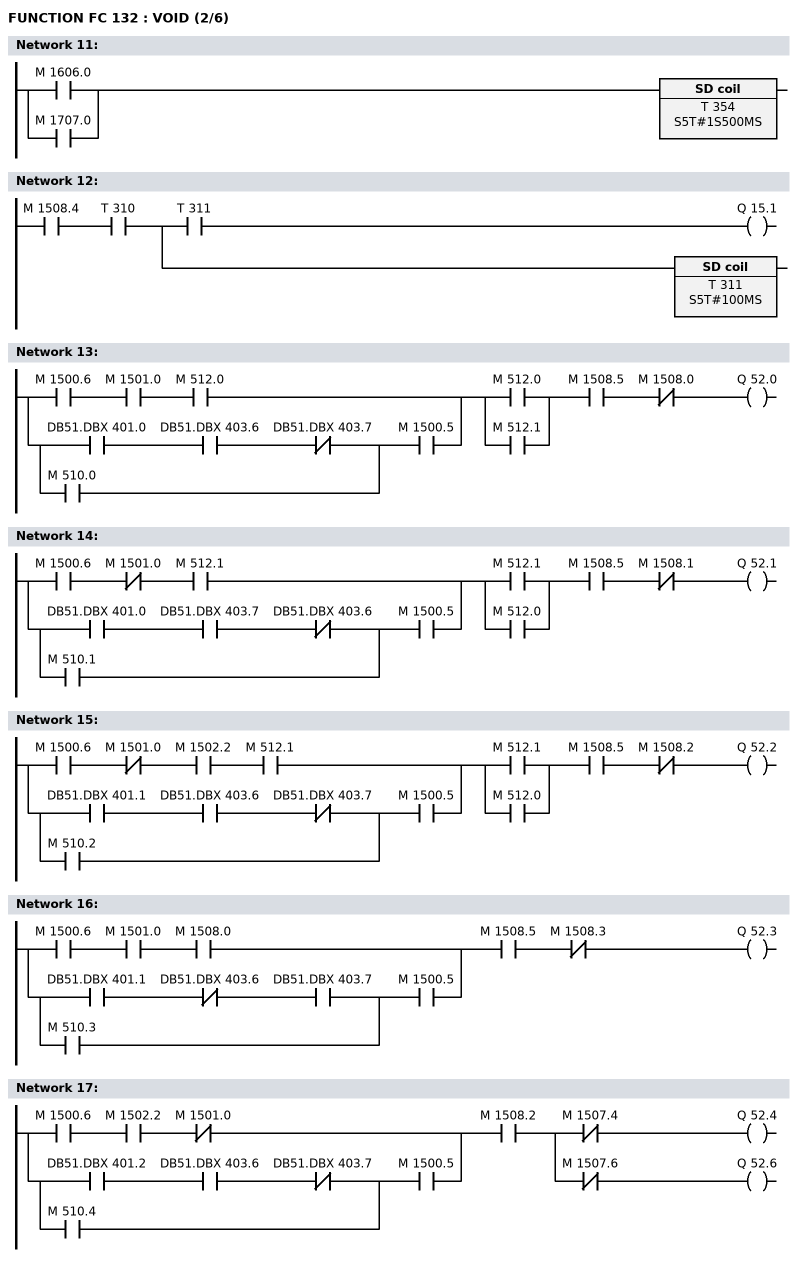

      O     M   1606.0;
      O     M   1707.0;
      L     S5T#1S500MS;
      SD    T    354;
NETWORK
TITLE =

      A     M   1508.4;
      A     T    310;
      =     L      0.0;
      A     L      0.0;
      A     T    311;
      =     Q     15.1;
      A     L      0.0;
      BLD   102;
      L     S5T#100MS;
      SD    T    311;
NETWORK
TITLE =

      A(    ;
      A     M   1500.6;
      A     M   1501.0;
      A     M    512.0;
      O     ;
      A(    ;
      A     DB51.DBX  401.0;
      A     DB51.DBX  403.6;
      AN    DB51.DBX  403.7;
      O     M    510.0;
      )     ;
      A     M   1500.5;
      )     ;
      A(    ;
      O     M    512.0;
      O     M    512.1;
      )     ;
      A     M   1508.5;
      AN    M   1508.0;
      =     Q     52.0;
NETWORK
TITLE =

      A(    ;
      A     M   1500.6;
      AN    M   1501.0;
      A     M    512.1;
      O     ;
      A(    ;
      A     DB51.DBX  401.0;
      A     DB51.DBX  403.7;
      AN    DB51.DBX  403.6;
      O     M    510.1;
      )     ;
      A     M   1500.5;
      )     ;
      A(    ;
      O     M    512.1;
      O     M    512.0;
      )     ;
      A     M   1508.5;
      AN    M   1508.1;
      =     Q     52.1;
NETWORK
TITLE =

      A(    ;
      A     M   1500.6;
      AN    M   1501.0;
      A     M   1502.2;
      A     M    512.1;
      O     ;
      A(    ;
      A     DB51.DBX  401.1;
      A     DB51.DBX  403.6;
      AN    DB51.DBX  403.7;
      O     M    510.2;
      )     ;
      A     M   1500.5;
      )     ;
      A(    ;
      O     M    512.1;
      O     M    512.0;
      )     ;
      A     M   1508.5;
      AN    M   1508.2;
      =     Q     52.2;
NETWORK
TITLE =

      A(    ;
      A     M   1500.6;
      A     M   1501.0;
      A     M   1508.0;
      O     ;
      A(    ;
      A     DB51.DBX  401.1;
      AN    DB51.DBX  403.6;
      A     DB51.DBX  403.7;
      O     M    510.3;
      )     ;
      A     M   1500.5;
      )     ;
      A     M   1508.5;
      AN    M   1508.3;
      =     Q     52.3;
NETWORK
TITLE =

      A(    ;
      A     M   1500.6;
      A     M   1502.2;
      AN    M   1501.0;
      O     ;
      A(    ;
      A     DB51.DBX  401.2;
      A     DB51.DBX  403.6;
      AN    DB51.DBX  403.7;
      O     M    510.4;
      )     ;
      A     M   1500.5;
      )     ;
      A     M   1508.2;
      =     L      0.0;
      A     L      0.0;
      AN    M   1507.4;
      =     Q     52.4;
      A     L      0.0;
      AN    M   1507.6;
      =     Q     52.6;
NETWORK
TITLE =
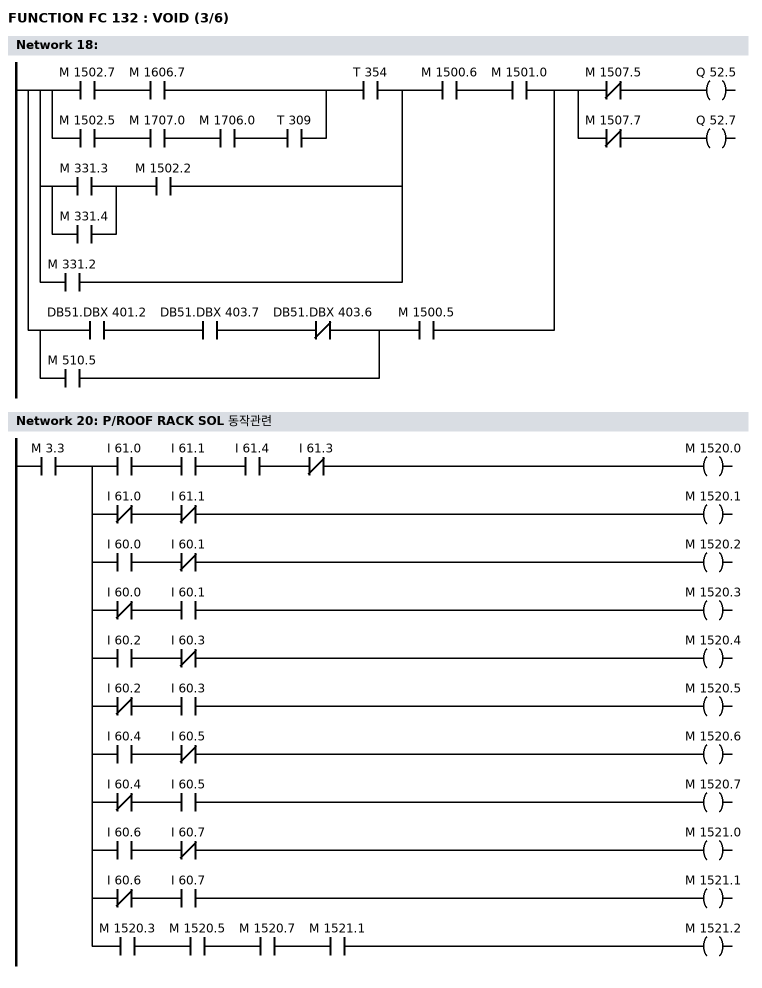

      A(    ;
      A(    ;
      A     M   1502.7;
      A     M   1606.7;
      O     ;
      A     M   1502.5;
      A     M   1707.0;
      A     M   1706.0;
      A     T    309;
      )     ;
      A     T    354;
      O     ;
      A(    ;
      O     M    331.3;
      O     M    331.4;
      )     ;
      A     M   1502.2;
      O     M    331.2;
      )     ;
      A     M   1500.6;
      A     M   1501.0;
      O     ;
      A(    ;
      A     DB51.DBX  401.2;
      A     DB51.DBX  403.7;
      AN    DB51.DBX  403.6;
      O     M    510.5;
      )     ;
      A     M   1500.5;
      =     L      0.0;
      A     L      0.0;
      AN    M   1507.5;
      =     Q     52.5;
      A     L      0.0;
      AN    M   1507.7;
      =     Q     52.7;
NETWORK
TITLE =

NETWORK
TITLE =P/ROOF RACK SOL 동작관련

      A     M      3.3;
      =     L      0.0;
      A     L      0.0;
      A     I     61.0;
      A     I     61.1;
      A     I     61.4;
      AN    I     61.3;
      =     M   1520.0;
      A     L      0.0;
      AN    I     61.0;
      AN    I     61.1;
      =     M   1520.1;
      A     L      0.0;
      A     I     60.0;
      AN    I     60.1;
      =     M   1520.2;
      A     L      0.0;
      AN    I     60.0;
      A     I     60.1;
      =     M   1520.3;
      A     L      0.0;
      A     I     60.2;
      AN    I     60.3;
      =     M   1520.4;
      A     L      0.0;
      AN    I     60.2;
      A     I     60.3;
      =     M   1520.5;
      A     L      0.0;
      A     I     60.4;
      AN    I     60.5;
      =     M   1520.6;
      A     L      0.0;
      AN    I     60.4;
      A     I     60.5;
      =     M   1520.7;
      A     L      0.0;
      A     I     60.6;
      AN    I     60.7;
      =     M   1521.0;
      A     L      0.0;
      AN    I     60.6;
      A     I     60.7;
      =     M   1521.1;
      A     L      0.0;
      A     M   1520.3;
      A     M   1520.5;
      A     M   1520.7;
      A     M   1521.1;
      =     M   1521.2;
NETWORK
TITLE =
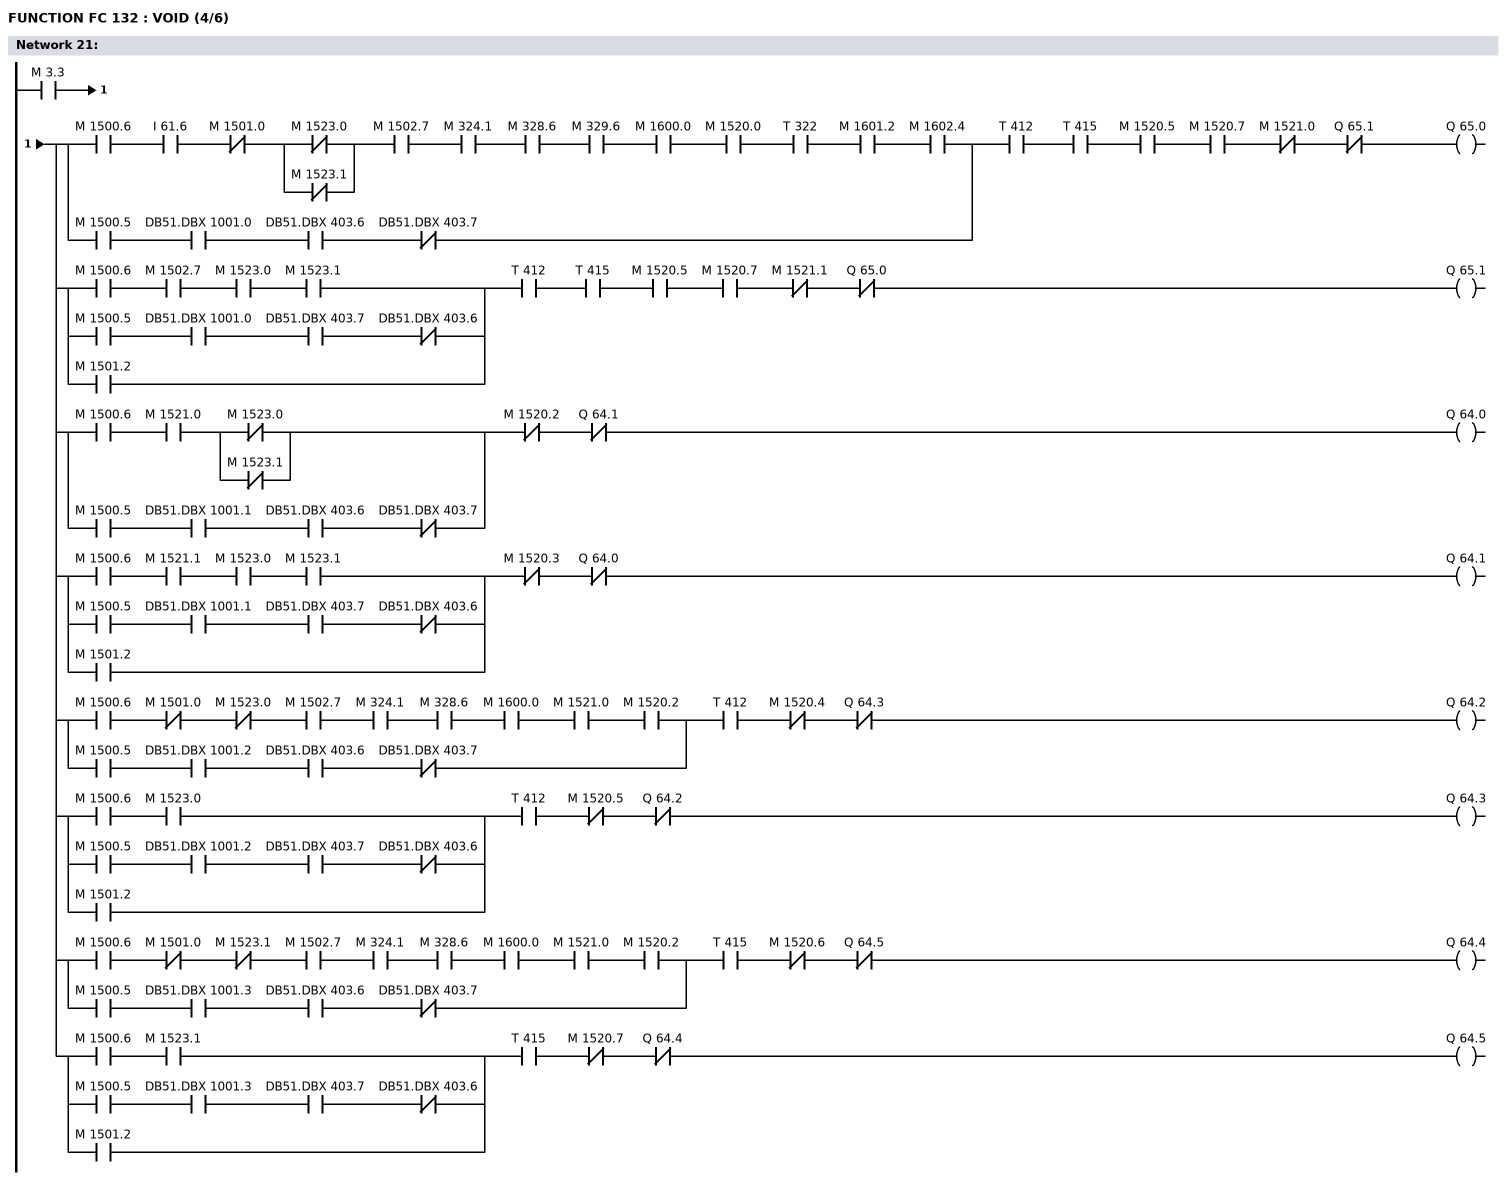

      A     M      3.3;
      =     L      0.0;
      A     L      0.0;
      A(    ;
      A     M   1500.6;
      A     I     61.6;
      AN    M   1501.0;
      A(    ;
      ON    M   1523.0;
      ON    M   1523.1;
      )     ;
      A     M   1502.7;
      A     M    324.1;
      A     M    328.6;
      A     M    329.6;
      A     M   1600.0;
      A     M   1520.0;
      A     T    322;
      A     M   1601.2;
      A     M   1602.4;
      O     ;
      A     M   1500.5;
      A     DB51.DBX 1001.0;
      A     DB51.DBX  403.6;
      AN    DB51.DBX  403.7;
      )     ;
      A     T    412;
      A     T    415;
      A     M   1520.5;
      A     M   1520.7;
      AN    M   1521.0;
      AN    Q     65.1;
      =     Q     65.0;
      A     L      0.0;
      A(    ;
      A     M   1500.6;
      A     M   1502.7;
      A     M   1523.0;
      A     M   1523.1;
      O     ;
      A     M   1500.5;
      A     DB51.DBX 1001.0;
      A     DB51.DBX  403.7;
      AN    DB51.DBX  403.6;
      O     M   1501.2;
      )     ;
      A     T    412;
      A     T    415;
      A     M   1520.5;
      A     M   1520.7;
      AN    M   1521.1;
      AN    Q     65.0;
      =     Q     65.1;
      A     L      0.0;
      A(    ;
      A     M   1500.6;
      A     M   1521.0;
      A(    ;
      ON    M   1523.0;
      ON    M   1523.1;
      )     ;
      O     ;
      A     M   1500.5;
      A     DB51.DBX 1001.1;
      A     DB51.DBX  403.6;
      AN    DB51.DBX  403.7;
      )     ;
      AN    M   1520.2;
      AN    Q     64.1;
      =     Q     64.0;
      A     L      0.0;
      A(    ;
      A     M   1500.6;
      A     M   1521.1;
      A     M   1523.0;
      A     M   1523.1;
      O     ;
      A     M   1500.5;
      A     DB51.DBX 1001.1;
      A     DB51.DBX  403.7;
      AN    DB51.DBX  403.6;
      O     M   1501.2;
      )     ;
      AN    M   1520.3;
      AN    Q     64.0;
      =     Q     64.1;
      A     L      0.0;
      A(    ;
      A     M   1500.6;
      AN    M   1501.0;
      AN    M   1523.0;
      A     M   1502.7;
      A     M    324.1;
      A     M    328.6;
      A     M   1600.0;
      A     M   1521.0;
      A     M   1520.2;
      O     ;
      A     M   1500.5;
      A     DB51.DBX 1001.2;
      A     DB51.DBX  403.6;
      AN    DB51.DBX  403.7;
      )     ;
      A     T    412;
      AN    M   1520.4;
      AN    Q     64.3;
      =     Q     64.2;
      A     L      0.0;
      A(    ;
      A     M   1500.6;
      A     M   1523.0;
      O     ;
      A     M   1500.5;
      A     DB51.DBX 1001.2;
      A     DB51.DBX  403.7;
      AN    DB51.DBX  403.6;
      O     M   1501.2;
      )     ;
      A     T    412;
      AN    M   1520.5;
      AN    Q     64.2;
      =     Q     64.3;
      A     L      0.0;
      A(    ;
      A     M   1500.6;
      AN    M   1501.0;
      AN    M   1523.1;
      A     M   1502.7;
      A     M    324.1;
      A     M    328.6;
      A     M   1600.0;
      A     M   1521.0;
      A     M   1520.2;
      O     ;
      A     M   1500.5;
      A     DB51.DBX 1001.3;
      A     DB51.DBX  403.6;
      AN    DB51.DBX  403.7;
      )     ;
      A     T    415;
      AN    M   1520.6;
      AN    Q     64.5;
      =     Q     64.4;
      A     L      0.0;
      A(    ;
      A     M   1500.6;
      A     M   1523.1;
      O     ;
      A     M   1500.5;
      A     DB51.DBX 1001.3;
      A     DB51.DBX  403.7;
      AN    DB51.DBX  403.6;
      O     M   1501.2;
      )     ;
      A     T    415;
      AN    M   1520.7;
      AN    Q     64.4;
      =     Q     64.5;
NETWORK
TITLE =
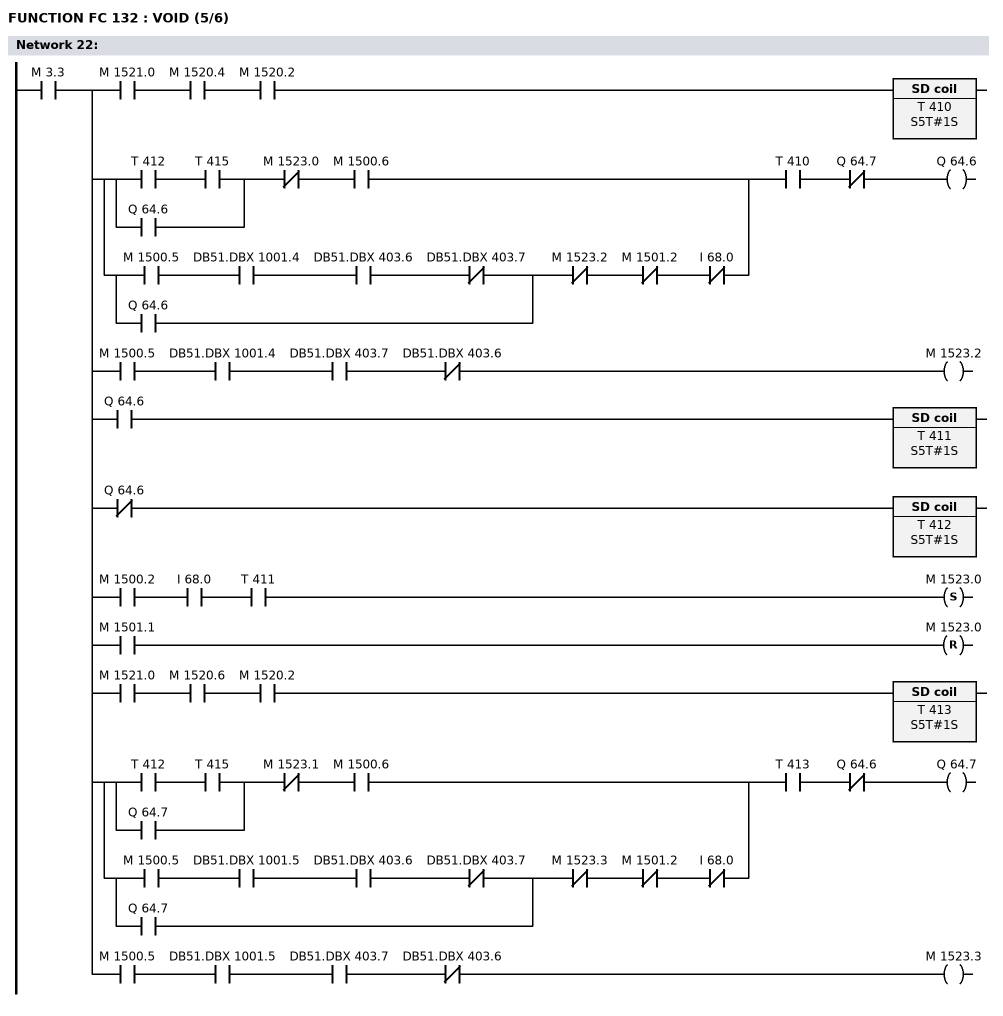

      A     M      3.3;
      =     L      0.0;
      A     L      0.0;
      A     M   1521.0;
      A     M   1520.4;
      A     M   1520.2;
      L     S5T#1S;
      SD    T    410;
      A     L      0.0;
      A(    ;
      A(    ;
      A     T    412;
      A     T    415;
      O     Q     64.6;
      )     ;
      AN    M   1523.0;
      A     M   1500.6;
      O     ;
      A(    ;
      A     M   1500.5;
      A     DB51.DBX 1001.4;
      A     DB51.DBX  403.6;
      AN    DB51.DBX  403.7;
      O     Q     64.6;
      )     ;
      AN    M   1523.2;
      AN    M   1501.2;
      AN    I     68.0;
      )     ;
      A     T    410;
      AN    Q     64.7;
      =     Q     64.6;
      A     L      0.0;
      A     M   1500.5;
      A     DB51.DBX 1001.4;
      A     DB51.DBX  403.7;
      AN    DB51.DBX  403.6;
      =     M   1523.2;
      A     L      0.0;
      A     Q     64.6;
      L     S5T#1S;
      SD    T    411;
      A     L      0.0;
      AN    Q     64.6;
      L     S5T#1S;
      SD    T    412;
      A     L      0.0;
      A     M   1500.2;
      A     I     68.0;
      A     T    411;
      S     M   1523.0;
      A     L      0.0;
      A     M   1501.1;
      R     M   1523.0;
      A     L      0.0;
      A     M   1521.0;
      A     M   1520.6;
      A     M   1520.2;
      L     S5T#1S;
      SD    T    413;
      A     L      0.0;
      A(    ;
      A(    ;
      A     T    412;
      A     T    415;
      O     Q     64.7;
      )     ;
      AN    M   1523.1;
      A     M   1500.6;
      O     ;
      A(    ;
      A     M   1500.5;
      A     DB51.DBX 1001.5;
      A     DB51.DBX  403.6;
      AN    DB51.DBX  403.7;
      O     Q     64.7;
      )     ;
      AN    M   1523.3;
      AN    M   1501.2;
      AN    I     68.0;
      )     ;
      A     T    413;
      AN    Q     64.6;
      =     Q     64.7;
      A     L      0.0;
      A     M   1500.5;
      A     DB51.DBX 1001.5;
      A     DB51.DBX  403.7;
      AN    DB51.DBX  403.6;
      =     M   1523.3;
NETWORK
TITLE =
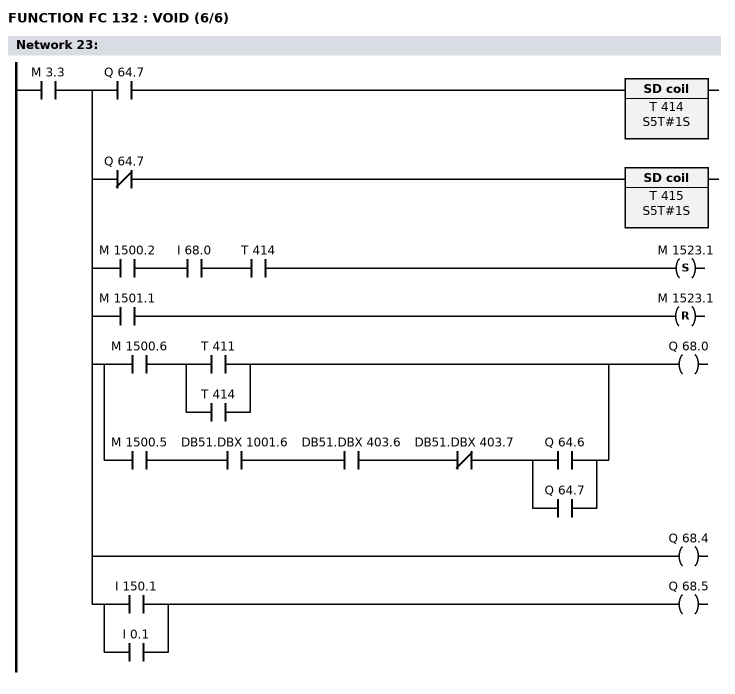

      A     M      3.3;
      =     L      0.0;
      A     L      0.0;
      A     Q     64.7;
      L     S5T#1S;
      SD    T    414;
      A     L      0.0;
      AN    Q     64.7;
      L     S5T#1S;
      SD    T    415;
      A     L      0.0;
      A     M   1500.2;
      A     I     68.0;
      A     T    414;
      S     M   1523.1;
      A     L      0.0;
      A     M   1501.1;
      R     M   1523.1;
      A     L      0.0;
      A(    ;
      A     M   1500.6;
      A(    ;
      O     T    411;
      O     T    414;
      )     ;
      O     ;
      A     M   1500.5;
      A     DB51.DBX 1001.6;
      A     DB51.DBX  403.6;
      AN    DB51.DBX  403.7;
      A(    ;
      O     Q     64.6;
      O     Q     64.7;
      )     ;
      )     ;
      =     Q     68.0;
      A     L      0.0;
      BLD   102;
      =     Q     68.4;
      A     L      0.0;
      A(    ;
      O     I    150.1;
      O     I      0.1;
      )     ;
      =     Q     68.5;
END_FUNCTION

FUNCTION_BLOCK FB 133
TITLE =
VERSION : 0.1


VAR
  S703_LM_DC_PIN : FB 424;
  S703_LM_DC_1ST_CLAMP1 : FB 424;
  S703_LM_DC_1ST_CLAMP2 : FB 424;
  S703_LM_DC_1ST_CLAMP3 : FB 424;
  S703_LM_DC_1ST_CLAMP4 : FB 424;
  S703_LM_DC_2ND_CLAMP1 : FB 424;
  S703_LM_DC_2ND_CLAMP2 : FB 424;
  S703_LM_DC_2ND_CLAMP3 : FB 424;
  S703_LM_DC_2ND_CLAMP4 : FB 424;
  S703_LM_DC_2ND_CLAMP5 : FB 424;
  S703_LM_DC_STK_PIN : FB 424;
  S703_LM_DC_OTR_CLAMP : FB 424;
  S703_LM_DC_ASSY_CLAMP : FB 424;
  S703_LM_DC_FF_PIN : FB 424;
  S703_LM_DC_FF_CLAMP : FB 424;
  S703_LM_DC_2ND_CLAMP6 : FB 424;
  S703_LM_DC_2ND_CLAMP7 : FB 424;
  S703_LM_DC_1ST_CLAMP5 : FB 424;
END_VAR
BEGIN
NETWORK
TITLE =
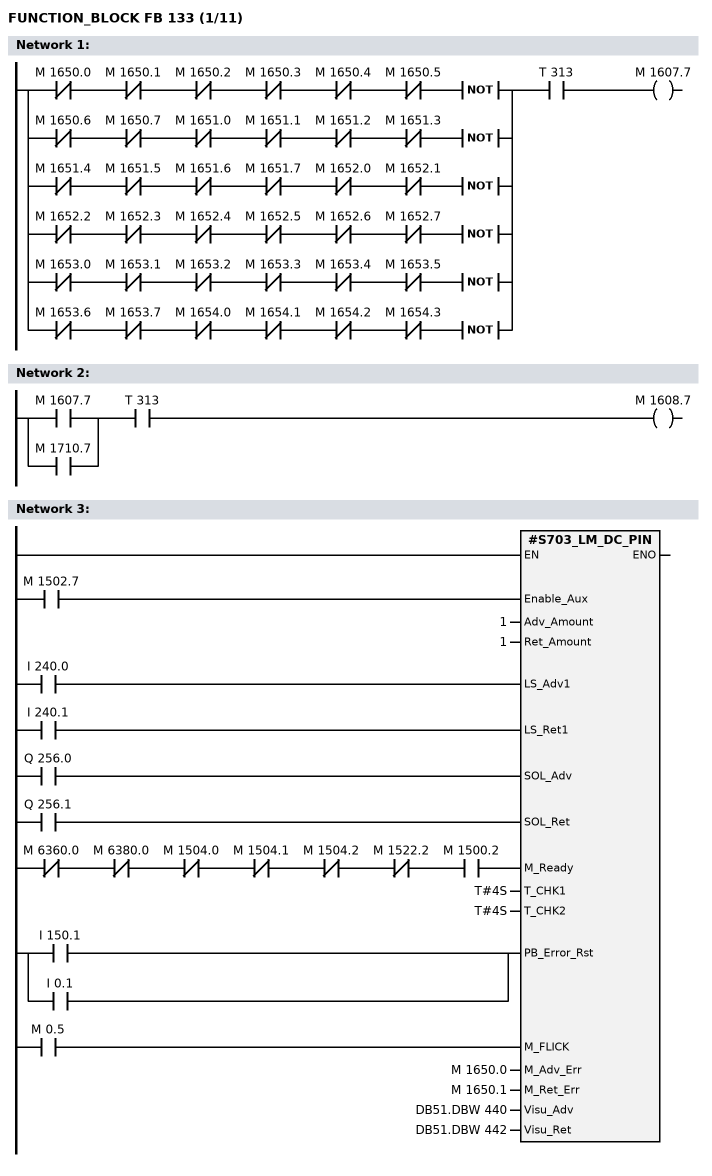

      A(    ;
      AN    M   1650.0;
      AN    M   1650.1;
      AN    M   1650.2;
      AN    M   1650.3;
      AN    M   1650.4;
      AN    M   1650.5;
      NOT   ;
      O(    ;
      AN    M   1650.6;
      AN    M   1650.7;
      AN    M   1651.0;
      AN    M   1651.1;
      AN    M   1651.2;
      AN    M   1651.3;
      NOT   ;
      )     ;
      O(    ;
      AN    M   1651.4;
      AN    M   1651.5;
      AN    M   1651.6;
      AN    M   1651.7;
      AN    M   1652.0;
      AN    M   1652.1;
      NOT   ;
      )     ;
      O(    ;
      AN    M   1652.2;
      AN    M   1652.3;
      AN    M   1652.4;
      AN    M   1652.5;
      AN    M   1652.6;
      AN    M   1652.7;
      NOT   ;
      )     ;
      O(    ;
      AN    M   1653.0;
      AN    M   1653.1;
      AN    M   1653.2;
      AN    M   1653.3;
      AN    M   1653.4;
      AN    M   1653.5;
      NOT   ;
      )     ;
      O(    ;
      AN    M   1653.6;
      AN    M   1653.7;
      AN    M   1654.0;
      AN    M   1654.1;
      AN    M   1654.2;
      AN    M   1654.3;
      NOT   ;
      )     ;
      )     ;
      A     T    313;
      =     M   1607.7;
NETWORK
TITLE =

      A(    ;
      O     M   1607.7;
      O     M   1710.7;
      )     ;
      A     T    313;
      =     M   1608.7;
NETWORK
TITLE =

      A     M   1502.7;
      =     L      0.0;
      BLD   103;
      A     I    240.0;
      =     L      0.1;
      BLD   103;
      A     I    240.1;
      =     L      0.2;
      BLD   103;
      A     Q    256.0;
      =     L      1.1;
      BLD   103;
      A     Q    256.1;
      =     L      1.2;
      BLD   103;
      AN    M   6360.0;
      AN    M   6380.0;
      AN    M   1504.0;
      AN    M   1504.1;
      AN    M   1504.2;
      AN    M   1522.2;
      A     M   1500.2;
      =     L      1.3;
      BLD   103;
      A(    ;
      O     I    150.1;
      O     I      0.1;
      )     ;
      =     L      1.5;
      BLD   103;
      A     M      0.5;
      =     L      1.6;
      BLD   103;
      CALL #S703_LM_DC_PIN (
           Enable_Aux               := L      0.0,
           Adv_Amount               := 1,
           Ret_Amount               := 1,
           LS_Adv1                  := L      0.1,
           LS_Ret1                  := L      0.2,
           SOL_Adv                  := L      1.1,
           SOL_Ret                  := L      1.2,
           M_Ready                  := L      1.3,
           T_CHK1                   := T#4S,
           T_CHK2                   := T#4S,
           PB_Error_Rst             := L      1.5,
           M_FLICK                  := L      1.6,
           M_Adv_Err                := M   1650.0,
           M_Ret_Err                := M   1650.1,
           Visu_Adv                 := DB51.DBW  440,
           Visu_Ret                 := DB51.DBW  442);
      NOP   0;
NETWORK
TITLE =
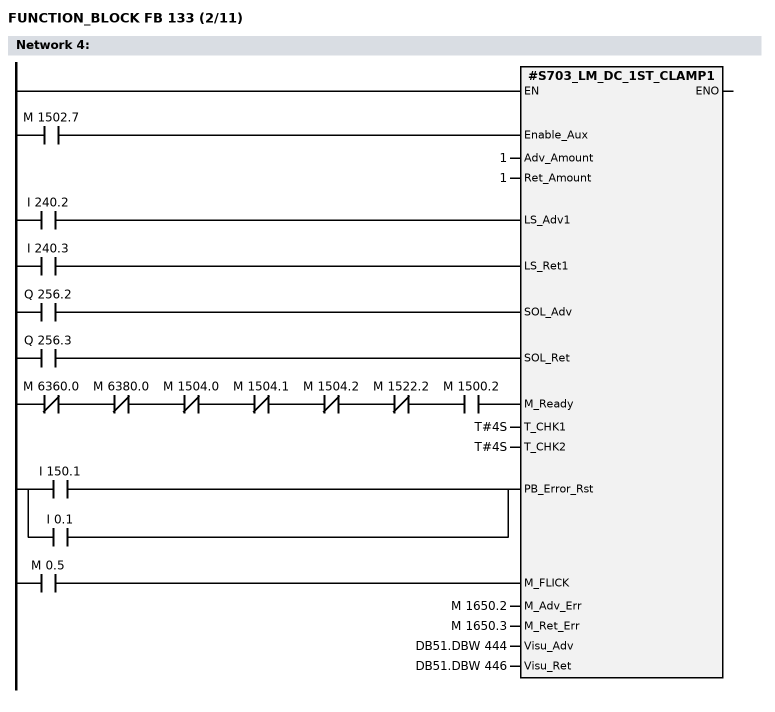

      A     M   1502.7;
      =     L      0.0;
      BLD   103;
      A     I    240.2;
      =     L      0.1;
      BLD   103;
      A     I    240.3;
      =     L      0.2;
      BLD   103;
      A     Q    256.2;
      =     L      1.1;
      BLD   103;
      A     Q    256.3;
      =     L      1.2;
      BLD   103;
      AN    M   6360.0;
      AN    M   6380.0;
      AN    M   1504.0;
      AN    M   1504.1;
      AN    M   1504.2;
      AN    M   1522.2;
      A     M   1500.2;
      =     L      1.3;
      BLD   103;
      A(    ;
      O     I    150.1;
      O     I      0.1;
      )     ;
      =     L      1.5;
      BLD   103;
      A     M      0.5;
      =     L      1.6;
      BLD   103;
      CALL #S703_LM_DC_1ST_CLAMP1 (
           Enable_Aux               := L      0.0,
           Adv_Amount               := 1,
           Ret_Amount               := 1,
           LS_Adv1                  := L      0.1,
           LS_Ret1                  := L      0.2,
           SOL_Adv                  := L      1.1,
           SOL_Ret                  := L      1.2,
           M_Ready                  := L      1.3,
           T_CHK1                   := T#4S,
           T_CHK2                   := T#4S,
           PB_Error_Rst             := L      1.5,
           M_FLICK                  := L      1.6,
           M_Adv_Err                := M   1650.2,
           M_Ret_Err                := M   1650.3,
           Visu_Adv                 := DB51.DBW  444,
           Visu_Ret                 := DB51.DBW  446);
      NOP   0;
NETWORK
TITLE =
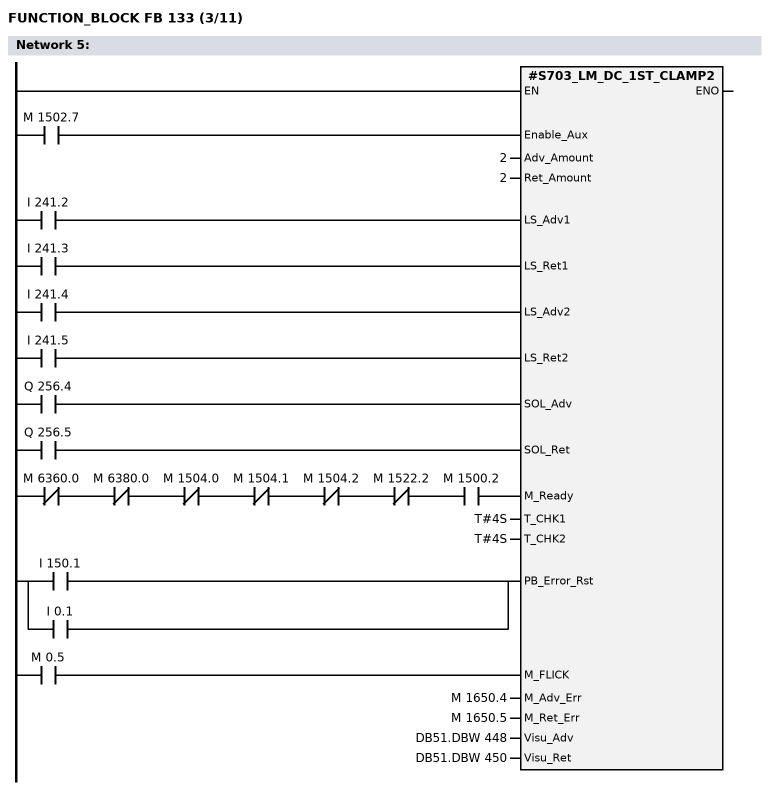

      A     M   1502.7;
      =     L      0.0;
      BLD   103;
      A     I    241.2;
      =     L      0.1;
      BLD   103;
      A     I    241.3;
      =     L      0.2;
      BLD   103;
      A     I    241.4;
      =     L      0.3;
      BLD   103;
      A     I    241.5;
      =     L      0.4;
      BLD   103;
      A     Q    256.4;
      =     L      1.1;
      BLD   103;
      A     Q    256.5;
      =     L      1.2;
      BLD   103;
      AN    M   6360.0;
      AN    M   6380.0;
      AN    M   1504.0;
      AN    M   1504.1;
      AN    M   1504.2;
      AN    M   1522.2;
      A     M   1500.2;
      =     L      1.3;
      BLD   103;
      A(    ;
      O     I    150.1;
      O     I      0.1;
      )     ;
      =     L      1.5;
      BLD   103;
      A     M      0.5;
      =     L      1.6;
      BLD   103;
      CALL #S703_LM_DC_1ST_CLAMP2 (
           Enable_Aux               := L      0.0,
           Adv_Amount               := 2,
           Ret_Amount               := 2,
           LS_Adv1                  := L      0.1,
           LS_Ret1                  := L      0.2,
           LS_Adv2                  := L      0.3,
           LS_Ret2                  := L      0.4,
           SOL_Adv                  := L      1.1,
           SOL_Ret                  := L      1.2,
           M_Ready                  := L      1.3,
           T_CHK1                   := T#4S,
           T_CHK2                   := T#4S,
           PB_Error_Rst             := L      1.5,
           M_FLICK                  := L      1.6,
           M_Adv_Err                := M   1650.4,
           M_Ret_Err                := M   1650.5,
           Visu_Adv                 := DB51.DBW  448,
           Visu_Ret                 := DB51.DBW  450);
      NOP   0;
NETWORK
TITLE =
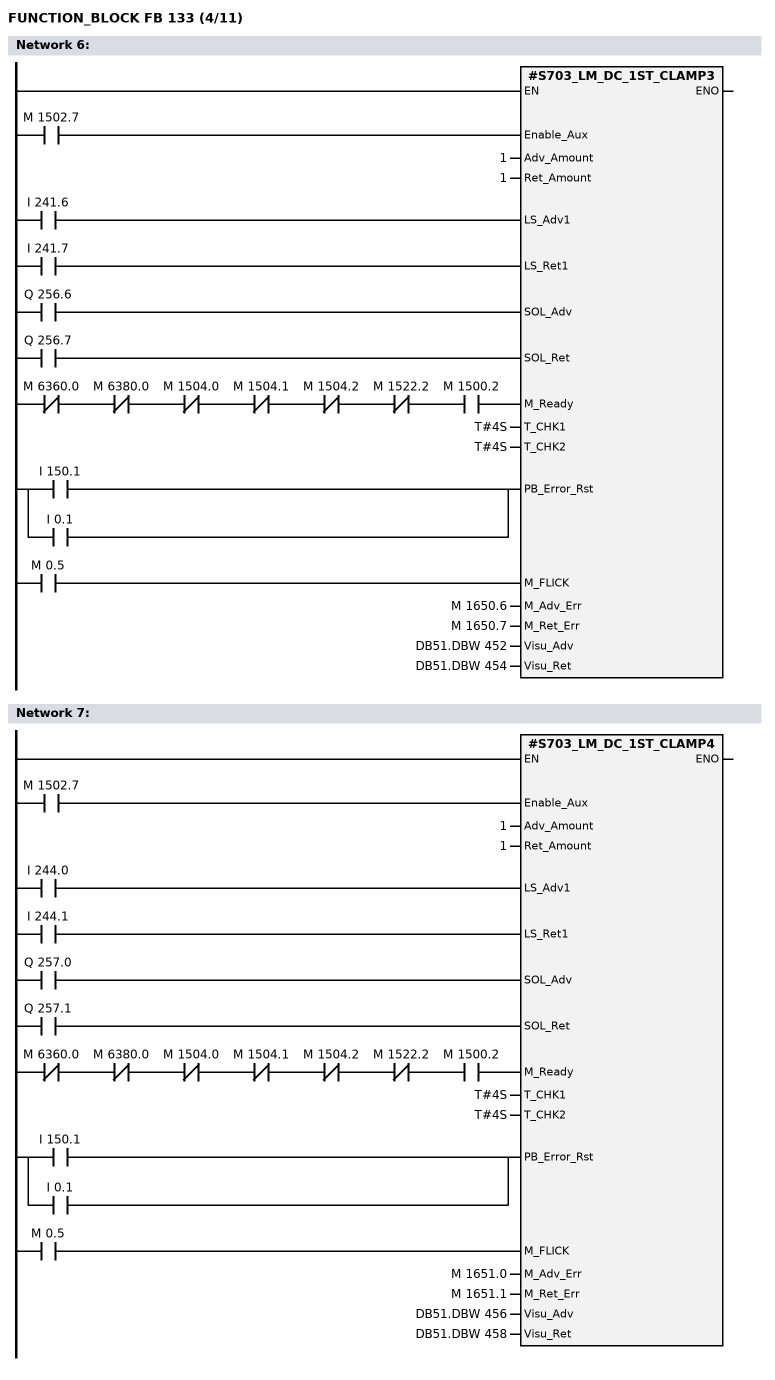

      A     M   1502.7;
      =     L      0.0;
      BLD   103;
      A     I    241.6;
      =     L      0.1;
      BLD   103;
      A     I    241.7;
      =     L      0.2;
      BLD   103;
      A     Q    256.6;
      =     L      1.1;
      BLD   103;
      A     Q    256.7;
      =     L      1.2;
      BLD   103;
      AN    M   6360.0;
      AN    M   6380.0;
      AN    M   1504.0;
      AN    M   1504.1;
      AN    M   1504.2;
      AN    M   1522.2;
      A     M   1500.2;
      =     L      1.3;
      BLD   103;
      A(    ;
      O     I    150.1;
      O     I      0.1;
      )     ;
      =     L      1.5;
      BLD   103;
      A     M      0.5;
      =     L      1.6;
      BLD   103;
      CALL #S703_LM_DC_1ST_CLAMP3 (
           Enable_Aux               := L      0.0,
           Adv_Amount               := 1,
           Ret_Amount               := 1,
           LS_Adv1                  := L      0.1,
           LS_Ret1                  := L      0.2,
           SOL_Adv                  := L      1.1,
           SOL_Ret                  := L      1.2,
           M_Ready                  := L      1.3,
           T_CHK1                   := T#4S,
           T_CHK2                   := T#4S,
           PB_Error_Rst             := L      1.5,
           M_FLICK                  := L      1.6,
           M_Adv_Err                := M   1650.6,
           M_Ret_Err                := M   1650.7,
           Visu_Adv                 := DB51.DBW  452,
           Visu_Ret                 := DB51.DBW  454);
      NOP   0;
NETWORK
TITLE =

      A     M   1502.7;
      =     L      0.0;
      BLD   103;
      A     I    244.0;
      =     L      0.1;
      BLD   103;
      A     I    244.1;
      =     L      0.2;
      BLD   103;
      A     Q    257.0;
      =     L      1.1;
      BLD   103;
      A     Q    257.1;
      =     L      1.2;
      BLD   103;
      AN    M   6360.0;
      AN    M   6380.0;
      AN    M   1504.0;
      AN    M   1504.1;
      AN    M   1504.2;
      AN    M   1522.2;
      A     M   1500.2;
      =     L      1.3;
      BLD   103;
      A(    ;
      O     I    150.1;
      O     I      0.1;
      )     ;
      =     L      1.5;
      BLD   103;
      A     M      0.5;
      =     L      1.6;
      BLD   103;
      CALL #S703_LM_DC_1ST_CLAMP4 (
           Enable_Aux               := L      0.0,
           Adv_Amount               := 1,
           Ret_Amount               := 1,
           LS_Adv1                  := L      0.1,
           LS_Ret1                  := L      0.2,
           SOL_Adv                  := L      1.1,
           SOL_Ret                  := L      1.2,
           M_Ready                  := L      1.3,
           T_CHK1                   := T#4S,
           T_CHK2                   := T#4S,
           PB_Error_Rst             := L      1.5,
           M_FLICK                  := L      1.6,
           M_Adv_Err                := M   1651.0,
           M_Ret_Err                := M   1651.1,
           Visu_Adv                 := DB51.DBW  456,
           Visu_Ret                 := DB51.DBW  458);
      NOP   0;
NETWORK
TITLE =
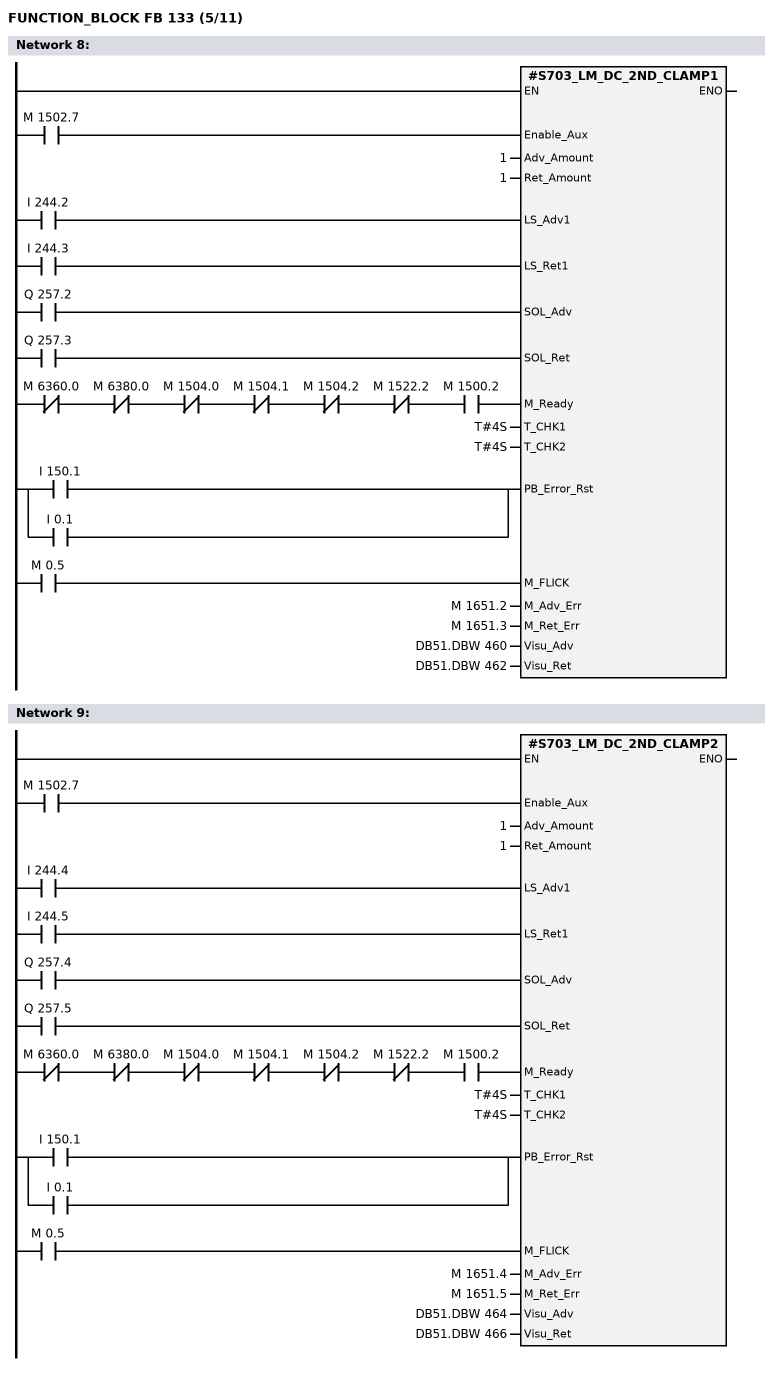

      A     M   1502.7;
      =     L      0.0;
      BLD   103;
      A     I    244.2;
      =     L      0.1;
      BLD   103;
      A     I    244.3;
      =     L      0.2;
      BLD   103;
      A     Q    257.2;
      =     L      1.1;
      BLD   103;
      A     Q    257.3;
      =     L      1.2;
      BLD   103;
      AN    M   6360.0;
      AN    M   6380.0;
      AN    M   1504.0;
      AN    M   1504.1;
      AN    M   1504.2;
      AN    M   1522.2;
      A     M   1500.2;
      =     L      1.3;
      BLD   103;
      A(    ;
      O     I    150.1;
      O     I      0.1;
      )     ;
      =     L      1.5;
      BLD   103;
      A     M      0.5;
      =     L      1.6;
      BLD   103;
      CALL #S703_LM_DC_2ND_CLAMP1 (
           Enable_Aux               := L      0.0,
           Adv_Amount               := 1,
           Ret_Amount               := 1,
           LS_Adv1                  := L      0.1,
           LS_Ret1                  := L      0.2,
           SOL_Adv                  := L      1.1,
           SOL_Ret                  := L      1.2,
           M_Ready                  := L      1.3,
           T_CHK1                   := T#4S,
           T_CHK2                   := T#4S,
           PB_Error_Rst             := L      1.5,
           M_FLICK                  := L      1.6,
           M_Adv_Err                := M   1651.2,
           M_Ret_Err                := M   1651.3,
           Visu_Adv                 := DB51.DBW  460,
           Visu_Ret                 := DB51.DBW  462);
      NOP   0;
NETWORK
TITLE =

      A     M   1502.7;
      =     L      0.0;
      BLD   103;
      A     I    244.4;
      =     L      0.1;
      BLD   103;
      A     I    244.5;
      =     L      0.2;
      BLD   103;
      A     Q    257.4;
      =     L      1.1;
      BLD   103;
      A     Q    257.5;
      =     L      1.2;
      BLD   103;
      AN    M   6360.0;
      AN    M   6380.0;
      AN    M   1504.0;
      AN    M   1504.1;
      AN    M   1504.2;
      AN    M   1522.2;
      A     M   1500.2;
      =     L      1.3;
      BLD   103;
      A(    ;
      O     I    150.1;
      O     I      0.1;
      )     ;
      =     L      1.5;
      BLD   103;
      A     M      0.5;
      =     L      1.6;
      BLD   103;
      CALL #S703_LM_DC_2ND_CLAMP2 (
           Enable_Aux               := L      0.0,
           Adv_Amount               := 1,
           Ret_Amount               := 1,
           LS_Adv1                  := L      0.1,
           LS_Ret1                  := L      0.2,
           SOL_Adv                  := L      1.1,
           SOL_Ret                  := L      1.2,
           M_Ready                  := L      1.3,
           T_CHK1                   := T#4S,
           T_CHK2                   := T#4S,
           PB_Error_Rst             := L      1.5,
           M_FLICK                  := L      1.6,
           M_Adv_Err                := M   1651.4,
           M_Ret_Err                := M   1651.5,
           Visu_Adv                 := DB51.DBW  464,
           Visu_Ret                 := DB51.DBW  466);
      NOP   0;
NETWORK
TITLE =
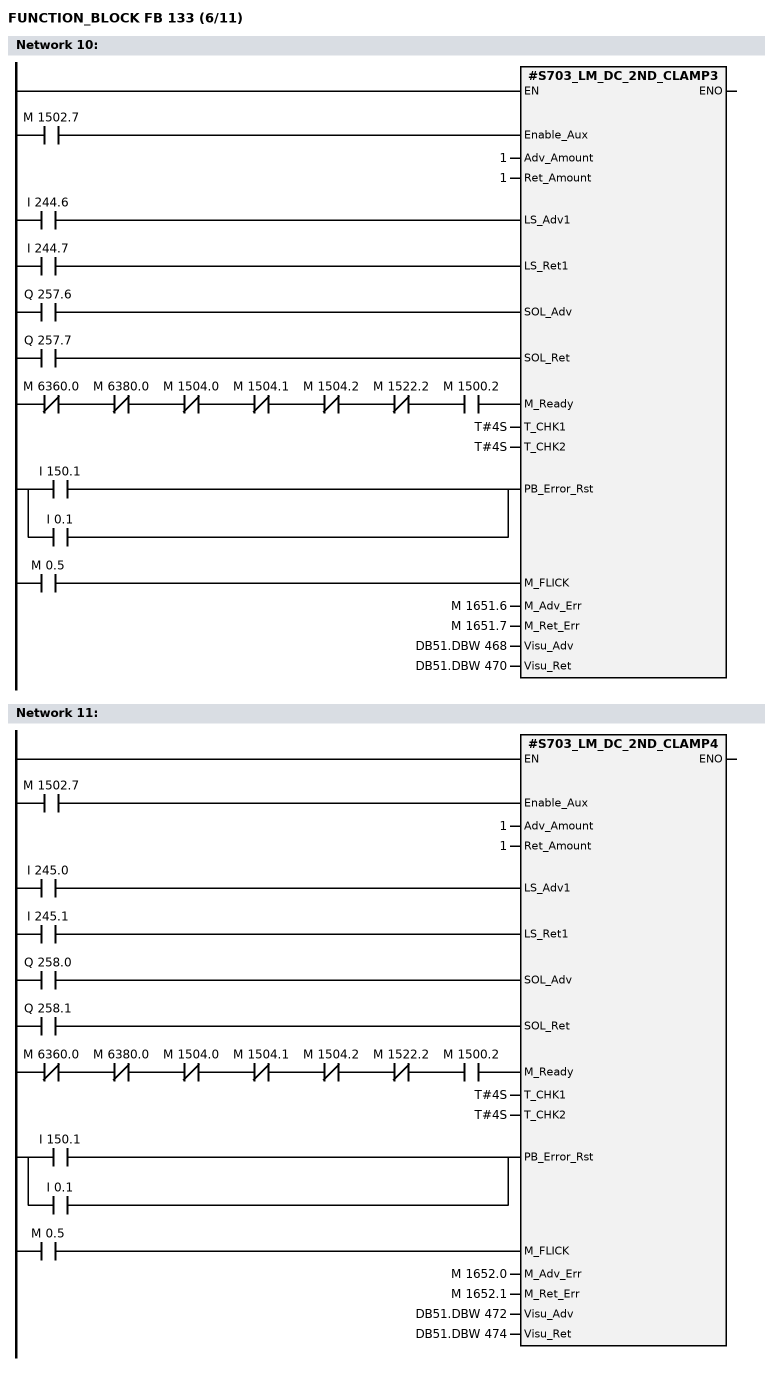

      A     M   1502.7;
      =     L      0.0;
      BLD   103;
      A     I    244.6;
      =     L      0.1;
      BLD   103;
      A     I    244.7;
      =     L      0.2;
      BLD   103;
      A     Q    257.6;
      =     L      1.1;
      BLD   103;
      A     Q    257.7;
      =     L      1.2;
      BLD   103;
      AN    M   6360.0;
      AN    M   6380.0;
      AN    M   1504.0;
      AN    M   1504.1;
      AN    M   1504.2;
      AN    M   1522.2;
      A     M   1500.2;
      =     L      1.3;
      BLD   103;
      A(    ;
      O     I    150.1;
      O     I      0.1;
      )     ;
      =     L      1.5;
      BLD   103;
      A     M      0.5;
      =     L      1.6;
      BLD   103;
      CALL #S703_LM_DC_2ND_CLAMP3 (
           Enable_Aux               := L      0.0,
           Adv_Amount               := 1,
           Ret_Amount               := 1,
           LS_Adv1                  := L      0.1,
           LS_Ret1                  := L      0.2,
           SOL_Adv                  := L      1.1,
           SOL_Ret                  := L      1.2,
           M_Ready                  := L      1.3,
           T_CHK1                   := T#4S,
           T_CHK2                   := T#4S,
           PB_Error_Rst             := L      1.5,
           M_FLICK                  := L      1.6,
           M_Adv_Err                := M   1651.6,
           M_Ret_Err                := M   1651.7,
           Visu_Adv                 := DB51.DBW  468,
           Visu_Ret                 := DB51.DBW  470);
      NOP   0;
NETWORK
TITLE =

      A     M   1502.7;
      =     L      0.0;
      BLD   103;
      A     I    245.0;
      =     L      0.1;
      BLD   103;
      A     I    245.1;
      =     L      0.2;
      BLD   103;
      A     Q    258.0;
      =     L      1.1;
      BLD   103;
      A     Q    258.1;
      =     L      1.2;
      BLD   103;
      AN    M   6360.0;
      AN    M   6380.0;
      AN    M   1504.0;
      AN    M   1504.1;
      AN    M   1504.2;
      AN    M   1522.2;
      A     M   1500.2;
      =     L      1.3;
      BLD   103;
      A(    ;
      O     I    150.1;
      O     I      0.1;
      )     ;
      =     L      1.5;
      BLD   103;
      A     M      0.5;
      =     L      1.6;
      BLD   103;
      CALL #S703_LM_DC_2ND_CLAMP4 (
           Enable_Aux               := L      0.0,
           Adv_Amount               := 1,
           Ret_Amount               := 1,
           LS_Adv1                  := L      0.1,
           LS_Ret1                  := L      0.2,
           SOL_Adv                  := L      1.1,
           SOL_Ret                  := L      1.2,
           M_Ready                  := L      1.3,
           T_CHK1                   := T#4S,
           T_CHK2                   := T#4S,
           PB_Error_Rst             := L      1.5,
           M_FLICK                  := L      1.6,
           M_Adv_Err                := M   1652.0,
           M_Ret_Err                := M   1652.1,
           Visu_Adv                 := DB51.DBW  472,
           Visu_Ret                 := DB51.DBW  474);
      NOP   0;
NETWORK
TITLE =
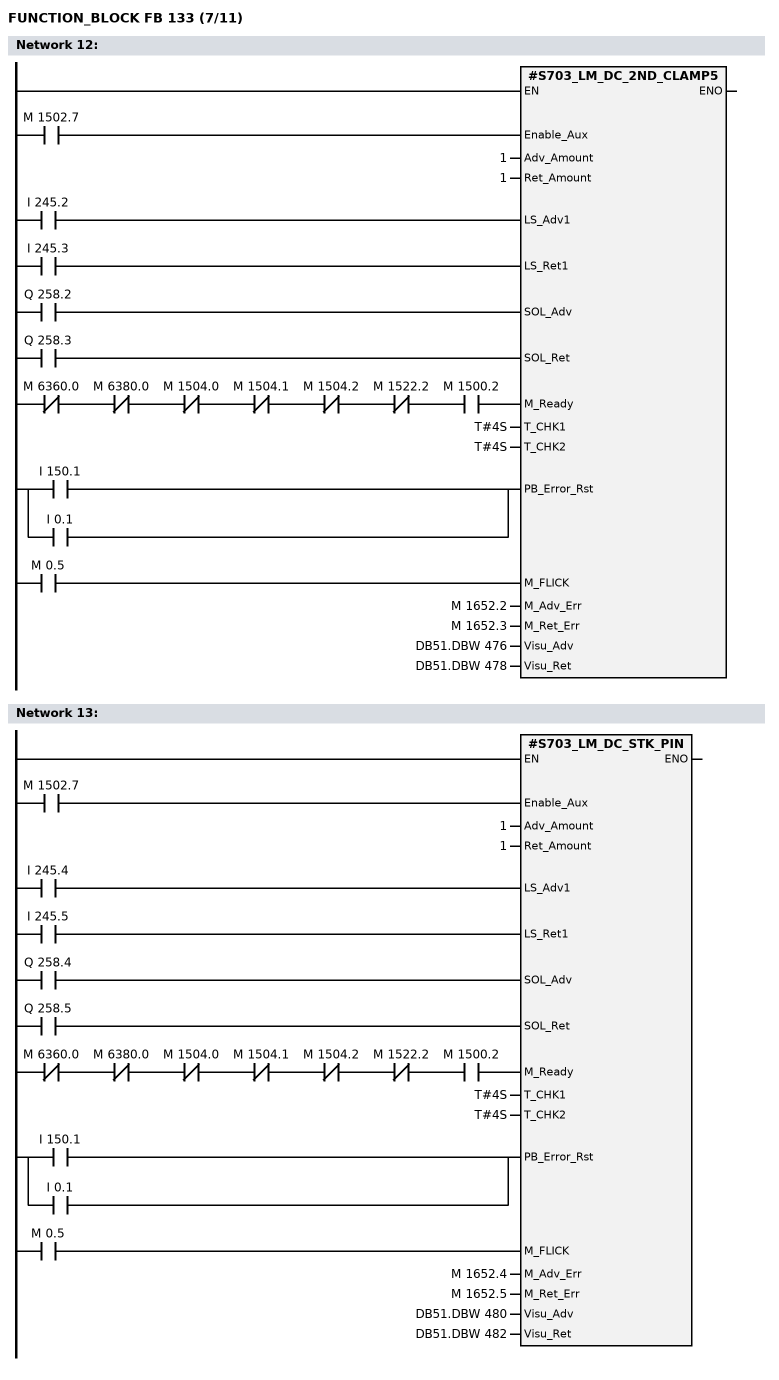

      A     M   1502.7;
      =     L      0.0;
      BLD   103;
      A     I    245.2;
      =     L      0.1;
      BLD   103;
      A     I    245.3;
      =     L      0.2;
      BLD   103;
      A     Q    258.2;
      =     L      1.1;
      BLD   103;
      A     Q    258.3;
      =     L      1.2;
      BLD   103;
      AN    M   6360.0;
      AN    M   6380.0;
      AN    M   1504.0;
      AN    M   1504.1;
      AN    M   1504.2;
      AN    M   1522.2;
      A     M   1500.2;
      =     L      1.3;
      BLD   103;
      A(    ;
      O     I    150.1;
      O     I      0.1;
      )     ;
      =     L      1.5;
      BLD   103;
      A     M      0.5;
      =     L      1.6;
      BLD   103;
      CALL #S703_LM_DC_2ND_CLAMP5 (
           Enable_Aux               := L      0.0,
           Adv_Amount               := 1,
           Ret_Amount               := 1,
           LS_Adv1                  := L      0.1,
           LS_Ret1                  := L      0.2,
           SOL_Adv                  := L      1.1,
           SOL_Ret                  := L      1.2,
           M_Ready                  := L      1.3,
           T_CHK1                   := T#4S,
           T_CHK2                   := T#4S,
           PB_Error_Rst             := L      1.5,
           M_FLICK                  := L      1.6,
           M_Adv_Err                := M   1652.2,
           M_Ret_Err                := M   1652.3,
           Visu_Adv                 := DB51.DBW  476,
           Visu_Ret                 := DB51.DBW  478);
      NOP   0;
NETWORK
TITLE =

      A     M   1502.7;
      =     L      0.0;
      BLD   103;
      A     I    245.4;
      =     L      0.1;
      BLD   103;
      A     I    245.5;
      =     L      0.2;
      BLD   103;
      A     Q    258.4;
      =     L      1.1;
      BLD   103;
      A     Q    258.5;
      =     L      1.2;
      BLD   103;
      AN    M   6360.0;
      AN    M   6380.0;
      AN    M   1504.0;
      AN    M   1504.1;
      AN    M   1504.2;
      AN    M   1522.2;
      A     M   1500.2;
      =     L      1.3;
      BLD   103;
      A(    ;
      O     I    150.1;
      O     I      0.1;
      )     ;
      =     L      1.5;
      BLD   103;
      A     M      0.5;
      =     L      1.6;
      BLD   103;
      CALL #S703_LM_DC_STK_PIN (
           Enable_Aux               := L      0.0,
           Adv_Amount               := 1,
           Ret_Amount               := 1,
           LS_Adv1                  := L      0.1,
           LS_Ret1                  := L      0.2,
           SOL_Adv                  := L      1.1,
           SOL_Ret                  := L      1.2,
           M_Ready                  := L      1.3,
           T_CHK1                   := T#4S,
           T_CHK2                   := T#4S,
           PB_Error_Rst             := L      1.5,
           M_FLICK                  := L      1.6,
           M_Adv_Err                := M   1652.4,
           M_Ret_Err                := M   1652.5,
           Visu_Adv                 := DB51.DBW  480,
           Visu_Ret                 := DB51.DBW  482);
      NOP   0;
NETWORK
TITLE =
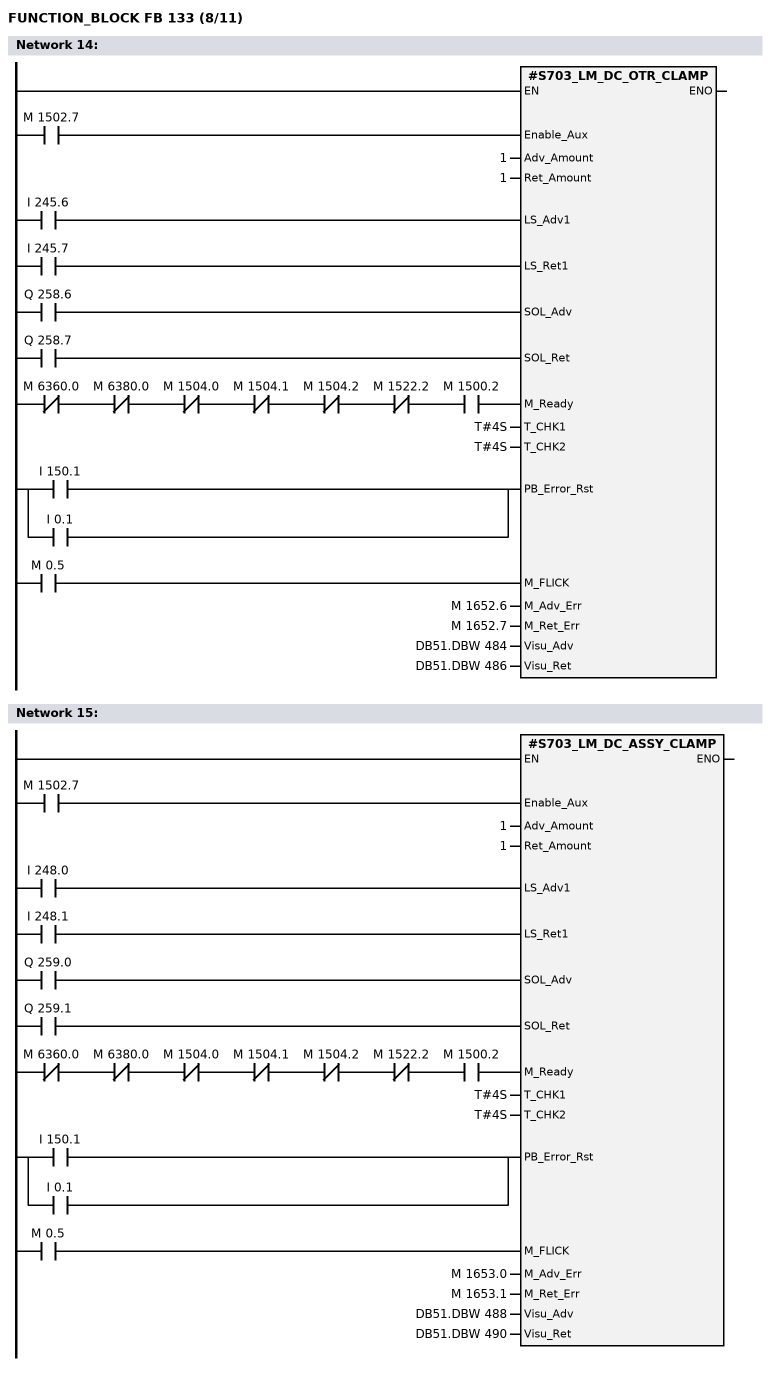

      A     M   1502.7;
      =     L      0.0;
      BLD   103;
      A     I    245.6;
      =     L      0.1;
      BLD   103;
      A     I    245.7;
      =     L      0.2;
      BLD   103;
      A     Q    258.6;
      =     L      1.1;
      BLD   103;
      A     Q    258.7;
      =     L      1.2;
      BLD   103;
      AN    M   6360.0;
      AN    M   6380.0;
      AN    M   1504.0;
      AN    M   1504.1;
      AN    M   1504.2;
      AN    M   1522.2;
      A     M   1500.2;
      =     L      1.3;
      BLD   103;
      A(    ;
      O     I    150.1;
      O     I      0.1;
      )     ;
      =     L      1.5;
      BLD   103;
      A     M      0.5;
      =     L      1.6;
      BLD   103;
      CALL #S703_LM_DC_OTR_CLAMP (
           Enable_Aux               := L      0.0,
           Adv_Amount               := 1,
           Ret_Amount               := 1,
           LS_Adv1                  := L      0.1,
           LS_Ret1                  := L      0.2,
           SOL_Adv                  := L      1.1,
           SOL_Ret                  := L      1.2,
           M_Ready                  := L      1.3,
           T_CHK1                   := T#4S,
           T_CHK2                   := T#4S,
           PB_Error_Rst             := L      1.5,
           M_FLICK                  := L      1.6,
           M_Adv_Err                := M   1652.6,
           M_Ret_Err                := M   1652.7,
           Visu_Adv                 := DB51.DBW  484,
           Visu_Ret                 := DB51.DBW  486);
      NOP   0;
NETWORK
TITLE =

      A     M   1502.7;
      =     L      0.0;
      BLD   103;
      A     I    248.0;
      =     L      0.1;
      BLD   103;
      A     I    248.1;
      =     L      0.2;
      BLD   103;
      A     Q    259.0;
      =     L      1.1;
      BLD   103;
      A     Q    259.1;
      =     L      1.2;
      BLD   103;
      AN    M   6360.0;
      AN    M   6380.0;
      AN    M   1504.0;
      AN    M   1504.1;
      AN    M   1504.2;
      AN    M   1522.2;
      A     M   1500.2;
      =     L      1.3;
      BLD   103;
      A(    ;
      O     I    150.1;
      O     I      0.1;
      )     ;
      =     L      1.5;
      BLD   103;
      A     M      0.5;
      =     L      1.6;
      BLD   103;
      CALL #S703_LM_DC_ASSY_CLAMP (
           Enable_Aux               := L      0.0,
           Adv_Amount               := 1,
           Ret_Amount               := 1,
           LS_Adv1                  := L      0.1,
           LS_Ret1                  := L      0.2,
           SOL_Adv                  := L      1.1,
           SOL_Ret                  := L      1.2,
           M_Ready                  := L      1.3,
           T_CHK1                   := T#4S,
           T_CHK2                   := T#4S,
           PB_Error_Rst             := L      1.5,
           M_FLICK                  := L      1.6,
           M_Adv_Err                := M   1653.0,
           M_Ret_Err                := M   1653.1,
           Visu_Adv                 := DB51.DBW  488,
           Visu_Ret                 := DB51.DBW  490);
      NOP   0;
NETWORK
TITLE =
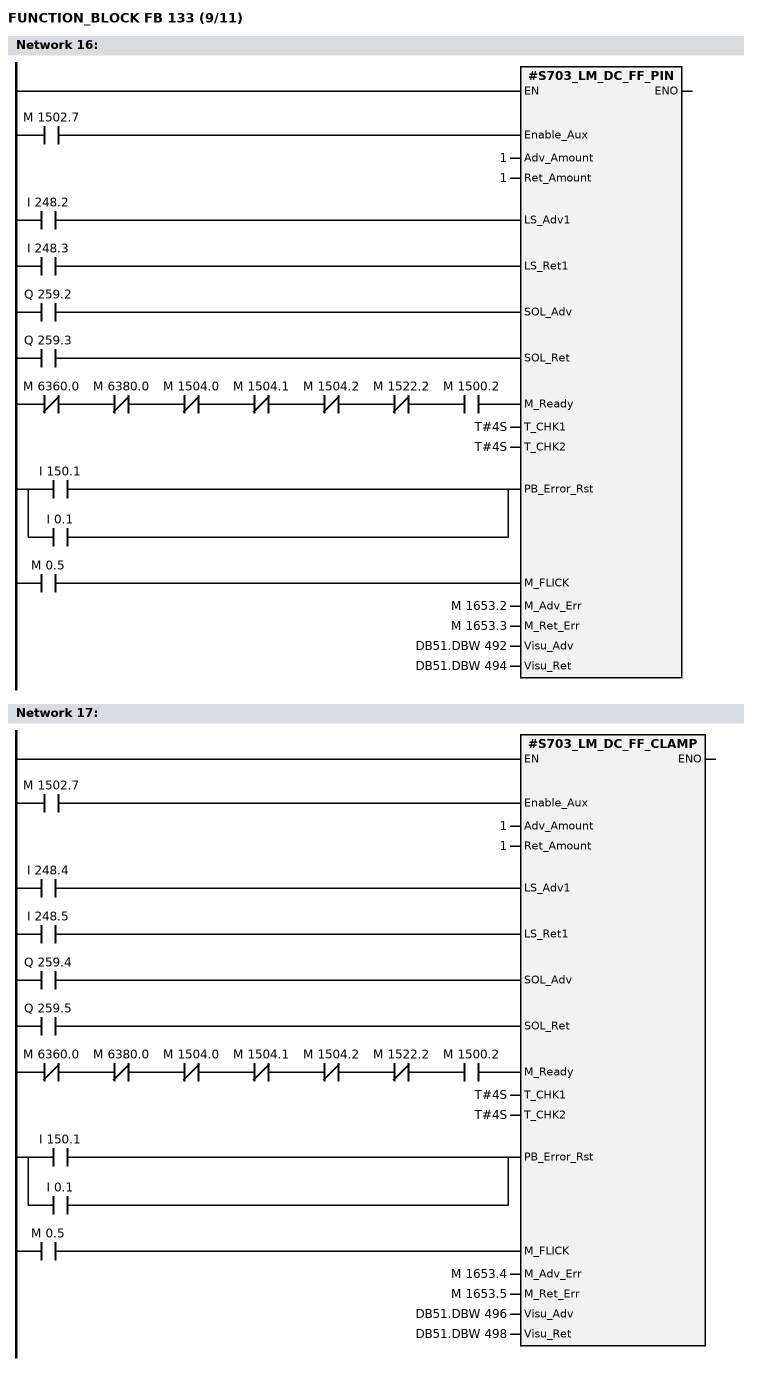

      A     M   1502.7;
      =     L      0.0;
      BLD   103;
      A     I    248.2;
      =     L      0.1;
      BLD   103;
      A     I    248.3;
      =     L      0.2;
      BLD   103;
      A     Q    259.2;
      =     L      1.1;
      BLD   103;
      A     Q    259.3;
      =     L      1.2;
      BLD   103;
      AN    M   6360.0;
      AN    M   6380.0;
      AN    M   1504.0;
      AN    M   1504.1;
      AN    M   1504.2;
      AN    M   1522.2;
      A     M   1500.2;
      =     L      1.3;
      BLD   103;
      A(    ;
      O     I    150.1;
      O     I      0.1;
      )     ;
      =     L      1.5;
      BLD   103;
      A     M      0.5;
      =     L      1.6;
      BLD   103;
      CALL #S703_LM_DC_FF_PIN (
           Enable_Aux               := L      0.0,
           Adv_Amount               := 1,
           Ret_Amount               := 1,
           LS_Adv1                  := L      0.1,
           LS_Ret1                  := L      0.2,
           SOL_Adv                  := L      1.1,
           SOL_Ret                  := L      1.2,
           M_Ready                  := L      1.3,
           T_CHK1                   := T#4S,
           T_CHK2                   := T#4S,
           PB_Error_Rst             := L      1.5,
           M_FLICK                  := L      1.6,
           M_Adv_Err                := M   1653.2,
           M_Ret_Err                := M   1653.3,
           Visu_Adv                 := DB51.DBW  492,
           Visu_Ret                 := DB51.DBW  494);
      NOP   0;
NETWORK
TITLE =

      A     M   1502.7;
      =     L      0.0;
      BLD   103;
      A     I    248.4;
      =     L      0.1;
      BLD   103;
      A     I    248.5;
      =     L      0.2;
      BLD   103;
      A     Q    259.4;
      =     L      1.1;
      BLD   103;
      A     Q    259.5;
      =     L      1.2;
      BLD   103;
      AN    M   6360.0;
      AN    M   6380.0;
      AN    M   1504.0;
      AN    M   1504.1;
      AN    M   1504.2;
      AN    M   1522.2;
      A     M   1500.2;
      =     L      1.3;
      BLD   103;
      A(    ;
      O     I    150.1;
      O     I      0.1;
      )     ;
      =     L      1.5;
      BLD   103;
      A     M      0.5;
      =     L      1.6;
      BLD   103;
      CALL #S703_LM_DC_FF_CLAMP (
           Enable_Aux               := L      0.0,
           Adv_Amount               := 1,
           Ret_Amount               := 1,
           LS_Adv1                  := L      0.1,
           LS_Ret1                  := L      0.2,
           SOL_Adv                  := L      1.1,
           SOL_Ret                  := L      1.2,
           M_Ready                  := L      1.3,
           T_CHK1                   := T#4S,
           T_CHK2                   := T#4S,
           PB_Error_Rst             := L      1.5,
           M_FLICK                  := L      1.6,
           M_Adv_Err                := M   1653.4,
           M_Ret_Err                := M   1653.5,
           Visu_Adv                 := DB51.DBW  496,
           Visu_Ret                 := DB51.DBW  498);
      NOP   0;
NETWORK
TITLE =
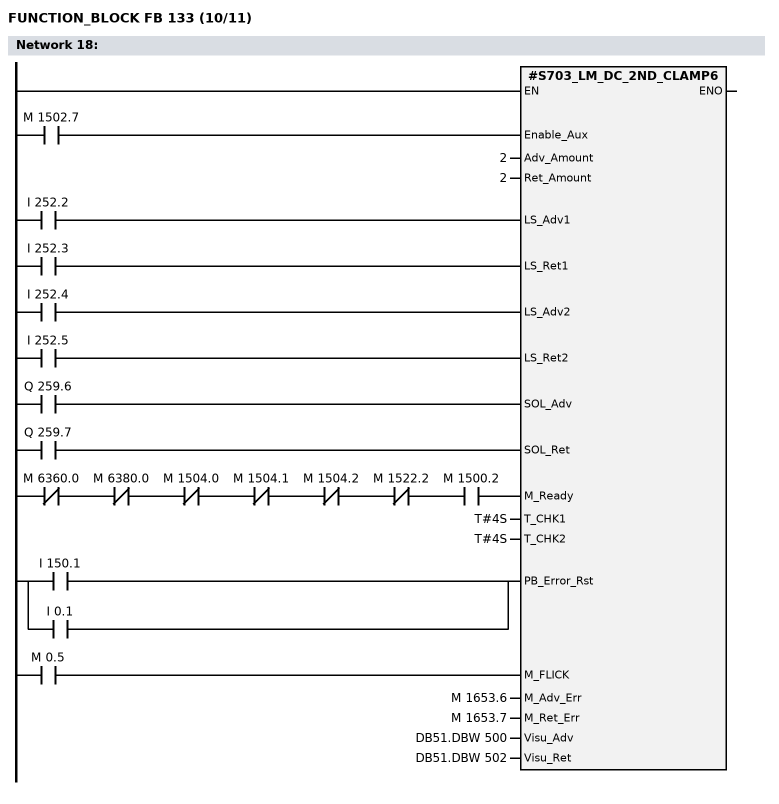

      A     M   1502.7;
      =     L      0.0;
      BLD   103;
      A     I    252.2;
      =     L      0.1;
      BLD   103;
      A     I    252.3;
      =     L      0.2;
      BLD   103;
      A     I    252.4;
      =     L      0.3;
      BLD   103;
      A     I    252.5;
      =     L      0.4;
      BLD   103;
      A     Q    259.6;
      =     L      1.1;
      BLD   103;
      A     Q    259.7;
      =     L      1.2;
      BLD   103;
      AN    M   6360.0;
      AN    M   6380.0;
      AN    M   1504.0;
      AN    M   1504.1;
      AN    M   1504.2;
      AN    M   1522.2;
      A     M   1500.2;
      =     L      1.3;
      BLD   103;
      A(    ;
      O     I    150.1;
      O     I      0.1;
      )     ;
      =     L      1.5;
      BLD   103;
      A     M      0.5;
      =     L      1.6;
      BLD   103;
      CALL #S703_LM_DC_2ND_CLAMP6 (
           Enable_Aux               := L      0.0,
           Adv_Amount               := 2,
           Ret_Amount               := 2,
           LS_Adv1                  := L      0.1,
           LS_Ret1                  := L      0.2,
           LS_Adv2                  := L      0.3,
           LS_Ret2                  := L      0.4,
           SOL_Adv                  := L      1.1,
           SOL_Ret                  := L      1.2,
           M_Ready                  := L      1.3,
           T_CHK1                   := T#4S,
           T_CHK2                   := T#4S,
           PB_Error_Rst             := L      1.5,
           M_FLICK                  := L      1.6,
           M_Adv_Err                := M   1653.6,
           M_Ret_Err                := M   1653.7,
           Visu_Adv                 := DB51.DBW  500,
           Visu_Ret                 := DB51.DBW  502);
      NOP   0;
NETWORK
TITLE =
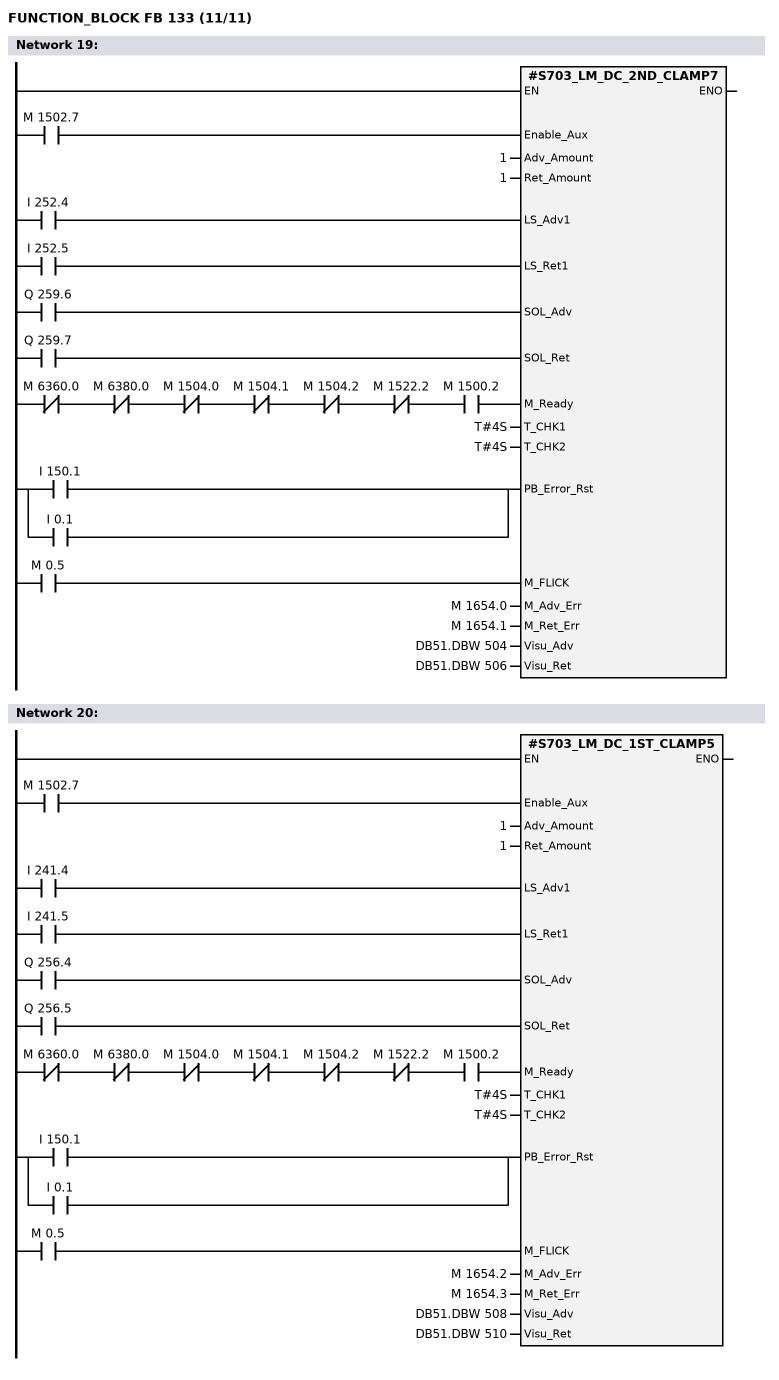

      A     M   1502.7;
      =     L      0.0;
      BLD   103;
      A     I    252.4;
      =     L      0.1;
      BLD   103;
      A     I    252.5;
      =     L      0.2;
      BLD   103;
      A     Q    259.6;
      =     L      1.1;
      BLD   103;
      A     Q    259.7;
      =     L      1.2;
      BLD   103;
      AN    M   6360.0;
      AN    M   6380.0;
      AN    M   1504.0;
      AN    M   1504.1;
      AN    M   1504.2;
      AN    M   1522.2;
      A     M   1500.2;
      =     L      1.3;
      BLD   103;
      A(    ;
      O     I    150.1;
      O     I      0.1;
      )     ;
      =     L      1.5;
      BLD   103;
      A     M      0.5;
      =     L      1.6;
      BLD   103;
      CALL #S703_LM_DC_2ND_CLAMP7 (
           Enable_Aux               := L      0.0,
           Adv_Amount               := 1,
           Ret_Amount               := 1,
           LS_Adv1                  := L      0.1,
           LS_Ret1                  := L      0.2,
           SOL_Adv                  := L      1.1,
           SOL_Ret                  := L      1.2,
           M_Ready                  := L      1.3,
           T_CHK1                   := T#4S,
           T_CHK2                   := T#4S,
           PB_Error_Rst             := L      1.5,
           M_FLICK                  := L      1.6,
           M_Adv_Err                := M   1654.0,
           M_Ret_Err                := M   1654.1,
           Visu_Adv                 := DB51.DBW  504,
           Visu_Ret                 := DB51.DBW  506);
      NOP   0;
NETWORK
TITLE =

      A     M   1502.7;
      =     L      0.0;
      BLD   103;
      A     I    241.4;
      =     L      0.1;
      BLD   103;
      A     I    241.5;
      =     L      0.2;
      BLD   103;
      A     Q    256.4;
      =     L      1.1;
      BLD   103;
      A     Q    256.5;
      =     L      1.2;
      BLD   103;
      AN    M   6360.0;
      AN    M   6380.0;
      AN    M   1504.0;
      AN    M   1504.1;
      AN    M   1504.2;
      AN    M   1522.2;
      A     M   1500.2;
      =     L      1.3;
      BLD   103;
      A(    ;
      O     I    150.1;
      O     I      0.1;
      )     ;
      =     L      1.5;
      BLD   103;
      A     M      0.5;
      =     L      1.6;
      BLD   103;
      CALL #S703_LM_DC_1ST_CLAMP5 (
           Enable_Aux               := L      0.0,
           Adv_Amount               := 1,
           Ret_Amount               := 1,
           LS_Adv1                  := L      0.1,
           LS_Ret1                  := L      0.2,
           SOL_Adv                  := L      1.1,
           SOL_Ret                  := L      1.2,
           M_Ready                  := L      1.3,
           T_CHK1                   := T#4S,
           T_CHK2                   := T#4S,
           PB_Error_Rst             := L      1.5,
           M_FLICK                  := L      1.6,
           M_Adv_Err                := M   1654.2,
           M_Ret_Err                := M   1654.3,
           Visu_Adv                 := DB51.DBW  508,
           Visu_Ret                 := DB51.DBW  510);
      NOP   0;
END_FUNCTION_BLOCK

DATA_BLOCK DB 133
TITLE =
VERSION : 0.0

 FB 133
BEGIN
   S703_LM_DC_PIN.Enable_Aux := FALSE;
   S703_LM_DC_PIN.Adv_Amount := 0;
   S703_LM_DC_PIN.Ret_Amount := 0;
   S703_LM_DC_PIN.LS_Adv1 := FALSE;
   S703_LM_DC_PIN.LS_Ret1 := FALSE;
   S703_LM_DC_PIN.LS_Adv2 := FALSE;
   S703_LM_DC_PIN.LS_Ret2 := FALSE;
   S703_LM_DC_PIN.LS_Adv3 := FALSE;
   S703_LM_DC_PIN.LS_Ret3 := FALSE;
   S703_LM_DC_PIN.LS_Adv4 := FALSE;
   S703_LM_DC_PIN.LS_Ret4 := FALSE;
   S703_LM_DC_PIN.SOL_Adv := FALSE;
   S703_LM_DC_PIN.SOL_Ret := FALSE;
   S703_LM_DC_PIN.M_Ready := FALSE;
   S703_LM_DC_PIN.T_CHK1 := T#0MS;
   S703_LM_DC_PIN.T_CHK2 := T#0MS;
   S703_LM_DC_PIN.PB_Lamp_CHK := FALSE;
   S703_LM_DC_PIN.PB_Error_Rst := FALSE;
   S703_LM_DC_PIN.M_FLICK := FALSE;
   S703_LM_DC_PIN.M_Adv_Err := FALSE;
   S703_LM_DC_PIN.M_Ret_Err := FALSE;
   S703_LM_DC_PIN.LP_Adv := FALSE;
   S703_LM_DC_PIN.LP_Ret := FALSE;
   S703_LM_DC_PIN.Visu_Adv := W#16#0;
   S703_LM_DC_PIN.Visu_Ret := W#16#0;
   S703_LM_DC_PIN.Error_T1.IN := FALSE;
   S703_LM_DC_PIN.Error_T1.PT := T#0MS;
   S703_LM_DC_PIN.Error_T1.Q := FALSE;
   S703_LM_DC_PIN.Error_T1.ET := T#0MS;
   S703_LM_DC_PIN.Error_T1.STATE := B#16#0;
   S703_LM_DC_PIN.Error_T1.STIME := T#0MS;
   S703_LM_DC_PIN.Error_T1.ATIME := T#0MS;
   S703_LM_DC_PIN.Error_T2.IN := FALSE;
   S703_LM_DC_PIN.Error_T2.PT := T#0MS;
   S703_LM_DC_PIN.Error_T2.Q := FALSE;
   S703_LM_DC_PIN.Error_T2.ET := T#0MS;
   S703_LM_DC_PIN.Error_T2.STATE := B#16#0;
   S703_LM_DC_PIN.Error_T2.STIME := T#0MS;
   S703_LM_DC_PIN.Error_T2.ATIME := T#0MS;
   S703_LM_DC_PIN.CHK_Aux1 := FALSE;
   S703_LM_DC_PIN.CHK_Aux2 := FALSE;
   S703_LM_DC_PIN.Error_T1_DN := FALSE;
   S703_LM_DC_PIN.Error_T2_DN := FALSE;
   S703_LM_DC_PIN.Adv_Memo := FALSE;
   S703_LM_DC_PIN.Visu_Adv_Arr[0] := FALSE;
   S703_LM_DC_PIN.Visu_Adv_Arr[1] := FALSE;
   S703_LM_DC_PIN.Visu_Adv_Arr[2] := FALSE;
   S703_LM_DC_PIN.Visu_Adv_Arr[3] := FALSE;
   S703_LM_DC_PIN.Visu_Adv_Arr[4] := FALSE;
   S703_LM_DC_PIN.Visu_Adv_Arr[5] := FALSE;
   S703_LM_DC_PIN.Visu_Adv_Arr[6] := FALSE;
   S703_LM_DC_PIN.Visu_Adv_Arr[7] := FALSE;
   S703_LM_DC_PIN.Visu_Adv_Arr[8] := FALSE;
   S703_LM_DC_PIN.Visu_Adv_Arr[9] := FALSE;
   S703_LM_DC_PIN.Visu_Adv_Arr[10] := FALSE;
   S703_LM_DC_PIN.Visu_Adv_Arr[11] := FALSE;
   S703_LM_DC_PIN.Visu_Adv_Arr[12] := FALSE;
   S703_LM_DC_PIN.Visu_Adv_Arr[13] := FALSE;
   S703_LM_DC_PIN.Visu_Adv_Arr[14] := FALSE;
   S703_LM_DC_PIN.Visu_Adv_Arr[15] := FALSE;
   S703_LM_DC_PIN.Visu_Ret_Arr[0] := FALSE;
   S703_LM_DC_PIN.Visu_Ret_Arr[1] := FALSE;
   S703_LM_DC_PIN.Visu_Ret_Arr[2] := FALSE;
   S703_LM_DC_PIN.Visu_Ret_Arr[3] := FALSE;
   S703_LM_DC_PIN.Visu_Ret_Arr[4] := FALSE;
   S703_LM_DC_PIN.Visu_Ret_Arr[5] := FALSE;
   S703_LM_DC_PIN.Visu_Ret_Arr[6] := FALSE;
   S703_LM_DC_PIN.Visu_Ret_Arr[7] := FALSE;
   S703_LM_DC_PIN.Visu_Ret_Arr[8] := FALSE;
   S703_LM_DC_PIN.Visu_Ret_Arr[9] := FALSE;
   S703_LM_DC_PIN.Visu_Ret_Arr[10] := FALSE;
   S703_LM_DC_PIN.Visu_Ret_Arr[11] := FALSE;
   S703_LM_DC_PIN.Visu_Ret_Arr[12] := FALSE;
   S703_LM_DC_PIN.Visu_Ret_Arr[13] := FALSE;
   S703_LM_DC_PIN.Visu_Ret_Arr[14] := FALSE;
   S703_LM_DC_PIN.Visu_Ret_Arr[15] := FALSE;
   S703_LM_DC_PIN.BLK_Move_Ret := 0;
   S703_LM_DC_PIN.Enable := FALSE;
   S703_LM_DC_PIN.Adv_End := FALSE;
   S703_LM_DC_PIN.Ret_End := FALSE;
   S703_LM_DC_1ST_CLAMP1.Enable_Aux := FALSE;
   S703_LM_DC_1ST_CLAMP1.Adv_Amount := 0;
   S703_LM_DC_1ST_CLAMP1.Ret_Amount := 0;
   S703_LM_DC_1ST_CLAMP1.LS_Adv1 := FALSE;
   S703_LM_DC_1ST_CLAMP1.LS_Ret1 := FALSE;
   S703_LM_DC_1ST_CLAMP1.LS_Adv2 := FALSE;
   S703_LM_DC_1ST_CLAMP1.LS_Ret2 := FALSE;
   S703_LM_DC_1ST_CLAMP1.LS_Adv3 := FALSE;
   S703_LM_DC_1ST_CLAMP1.LS_Ret3 := FALSE;
   S703_LM_DC_1ST_CLAMP1.LS_Adv4 := FALSE;
   S703_LM_DC_1ST_CLAMP1.LS_Ret4 := FALSE;
   S703_LM_DC_1ST_CLAMP1.SOL_Adv := FALSE;
   S703_LM_DC_1ST_CLAMP1.SOL_Ret := FALSE;
   S703_LM_DC_1ST_CLAMP1.M_Ready := FALSE;
   S703_LM_DC_1ST_CLAMP1.T_CHK1 := T#0MS;
   S703_LM_DC_1ST_CLAMP1.T_CHK2 := T#0MS;
   S703_LM_DC_1ST_CLAMP1.PB_Lamp_CHK := FALSE;
   S703_LM_DC_1ST_CLAMP1.PB_Error_Rst := FALSE;
   S703_LM_DC_1ST_CLAMP1.M_FLICK := FALSE;
   S703_LM_DC_1ST_CLAMP1.M_Adv_Err := FALSE;
   S703_LM_DC_1ST_CLAMP1.M_Ret_Err := FALSE;
   S703_LM_DC_1ST_CLAMP1.LP_Adv := FALSE;
   S703_LM_DC_1ST_CLAMP1.LP_Ret := FALSE;
   S703_LM_DC_1ST_CLAMP1.Visu_Adv := W#16#0;
   S703_LM_DC_1ST_CLAMP1.Visu_Ret := W#16#0;
   S703_LM_DC_1ST_CLAMP1.Error_T1.IN := FALSE;
   S703_LM_DC_1ST_CLAMP1.Error_T1.PT := T#0MS;
   S703_LM_DC_1ST_CLAMP1.Error_T1.Q := FALSE;
   S703_LM_DC_1ST_CLAMP1.Error_T1.ET := T#0MS;
   S703_LM_DC_1ST_CLAMP1.Error_T1.STATE := B#16#0;
   S703_LM_DC_1ST_CLAMP1.Error_T1.STIME := T#0MS;
   S703_LM_DC_1ST_CLAMP1.Error_T1.ATIME := T#0MS;
   S703_LM_DC_1ST_CLAMP1.Error_T2.IN := FALSE;
   S703_LM_DC_1ST_CLAMP1.Error_T2.PT := T#0MS;
   S703_LM_DC_1ST_CLAMP1.Error_T2.Q := FALSE;
   S703_LM_DC_1ST_CLAMP1.Error_T2.ET := T#0MS;
   S703_LM_DC_1ST_CLAMP1.Error_T2.STATE := B#16#0;
   S703_LM_DC_1ST_CLAMP1.Error_T2.STIME := T#0MS;
   S703_LM_DC_1ST_CLAMP1.Error_T2.ATIME := T#0MS;
   S703_LM_DC_1ST_CLAMP1.CHK_Aux1 := FALSE;
   S703_LM_DC_1ST_CLAMP1.CHK_Aux2 := FALSE;
   S703_LM_DC_1ST_CLAMP1.Error_T1_DN := FALSE;
   S703_LM_DC_1ST_CLAMP1.Error_T2_DN := FALSE;
   S703_LM_DC_1ST_CLAMP1.Adv_Memo := FALSE;
   S703_LM_DC_1ST_CLAMP1.Visu_Adv_Arr[0] := FALSE;
   S703_LM_DC_1ST_CLAMP1.Visu_Adv_Arr[1] := FALSE;
   S703_LM_DC_1ST_CLAMP1.Visu_Adv_Arr[2] := FALSE;
   S703_LM_DC_1ST_CLAMP1.Visu_Adv_Arr[3] := FALSE;
   S703_LM_DC_1ST_CLAMP1.Visu_Adv_Arr[4] := FALSE;
   S703_LM_DC_1ST_CLAMP1.Visu_Adv_Arr[5] := FALSE;
   S703_LM_DC_1ST_CLAMP1.Visu_Adv_Arr[6] := FALSE;
   S703_LM_DC_1ST_CLAMP1.Visu_Adv_Arr[7] := FALSE;
   S703_LM_DC_1ST_CLAMP1.Visu_Adv_Arr[8] := FALSE;
   S703_LM_DC_1ST_CLAMP1.Visu_Adv_Arr[9] := FALSE;
   S703_LM_DC_1ST_CLAMP1.Visu_Adv_Arr[10] := FALSE;
   S703_LM_DC_1ST_CLAMP1.Visu_Adv_Arr[11] := FALSE;
   S703_LM_DC_1ST_CLAMP1.Visu_Adv_Arr[12] := FALSE;
   S703_LM_DC_1ST_CLAMP1.Visu_Adv_Arr[13] := FALSE;
   S703_LM_DC_1ST_CLAMP1.Visu_Adv_Arr[14] := FALSE;
   S703_LM_DC_1ST_CLAMP1.Visu_Adv_Arr[15] := FALSE;
   S703_LM_DC_1ST_CLAMP1.Visu_Ret_Arr[0] := FALSE;
   S703_LM_DC_1ST_CLAMP1.Visu_Ret_Arr[1] := FALSE;
   S703_LM_DC_1ST_CLAMP1.Visu_Ret_Arr[2] := FALSE;
   S703_LM_DC_1ST_CLAMP1.Visu_Ret_Arr[3] := FALSE;
   S703_LM_DC_1ST_CLAMP1.Visu_Ret_Arr[4] := FALSE;
   S703_LM_DC_1ST_CLAMP1.Visu_Ret_Arr[5] := FALSE;
   S703_LM_DC_1ST_CLAMP1.Visu_Ret_Arr[6] := FALSE;
   S703_LM_DC_1ST_CLAMP1.Visu_Ret_Arr[7] := FALSE;
   S703_LM_DC_1ST_CLAMP1.Visu_Ret_Arr[8] := FALSE;
   S703_LM_DC_1ST_CLAMP1.Visu_Ret_Arr[9] := FALSE;
   S703_LM_DC_1ST_CLAMP1.Visu_Ret_Arr[10] := FALSE;
   S703_LM_DC_1ST_CLAMP1.Visu_Ret_Arr[11] := FALSE;
   S703_LM_DC_1ST_CLAMP1.Visu_Ret_Arr[12] := FALSE;
   S703_LM_DC_1ST_CLAMP1.Visu_Ret_Arr[13] := FALSE;
   S703_LM_DC_1ST_CLAMP1.Visu_Ret_Arr[14] := FALSE;
   S703_LM_DC_1ST_CLAMP1.Visu_Ret_Arr[15] := FALSE;
   S703_LM_DC_1ST_CLAMP1.BLK_Move_Ret := 0;
   S703_LM_DC_1ST_CLAMP1.Enable := FALSE;
   S703_LM_DC_1ST_CLAMP1.Adv_End := FALSE;
   S703_LM_DC_1ST_CLAMP1.Ret_End := FALSE;
   S703_LM_DC_1ST_CLAMP2.Enable_Aux := FALSE;
   S703_LM_DC_1ST_CLAMP2.Adv_Amount := 0;
   S703_LM_DC_1ST_CLAMP2.Ret_Amount := 0;
   S703_LM_DC_1ST_CLAMP2.LS_Adv1 := FALSE;
   S703_LM_DC_1ST_CLAMP2.LS_Ret1 := FALSE;
   S703_LM_DC_1ST_CLAMP2.LS_Adv2 := FALSE;
   S703_LM_DC_1ST_CLAMP2.LS_Ret2 := FALSE;
   S703_LM_DC_1ST_CLAMP2.LS_Adv3 := FALSE;
   S703_LM_DC_1ST_CLAMP2.LS_Ret3 := FALSE;
   S703_LM_DC_1ST_CLAMP2.LS_Adv4 := FALSE;
   S703_LM_DC_1ST_CLAMP2.LS_Ret4 := FALSE;
   S703_LM_DC_1ST_CLAMP2.SOL_Adv := FALSE;
   S703_LM_DC_1ST_CLAMP2.SOL_Ret := FALSE;
   S703_LM_DC_1ST_CLAMP2.M_Ready := FALSE;
   S703_LM_DC_1ST_CLAMP2.T_CHK1 := T#0MS;
   S703_LM_DC_1ST_CLAMP2.T_CHK2 := T#0MS;
   S703_LM_DC_1ST_CLAMP2.PB_Lamp_CHK := FALSE;
   S703_LM_DC_1ST_CLAMP2.PB_Error_Rst := FALSE;
   S703_LM_DC_1ST_CLAMP2.M_FLICK := FALSE;
   S703_LM_DC_1ST_CLAMP2.M_Adv_Err := FALSE;
   S703_LM_DC_1ST_CLAMP2.M_Ret_Err := FALSE;
   S703_LM_DC_1ST_CLAMP2.LP_Adv := FALSE;
   S703_LM_DC_1ST_CLAMP2.LP_Ret := FALSE;
   S703_LM_DC_1ST_CLAMP2.Visu_Adv := W#16#0;
   S703_LM_DC_1ST_CLAMP2.Visu_Ret := W#16#0;
   S703_LM_DC_1ST_CLAMP2.Error_T1.IN := FALSE;
   S703_LM_DC_1ST_CLAMP2.Error_T1.PT := T#0MS;
   S703_LM_DC_1ST_CLAMP2.Error_T1.Q := FALSE;
   S703_LM_DC_1ST_CLAMP2.Error_T1.ET := T#0MS;
   S703_LM_DC_1ST_CLAMP2.Error_T1.STATE := B#16#0;
   S703_LM_DC_1ST_CLAMP2.Error_T1.STIME := T#0MS;
   S703_LM_DC_1ST_CLAMP2.Error_T1.ATIME := T#0MS;
   S703_LM_DC_1ST_CLAMP2.Error_T2.IN := FALSE;
   S703_LM_DC_1ST_CLAMP2.Error_T2.PT := T#0MS;
   S703_LM_DC_1ST_CLAMP2.Error_T2.Q := FALSE;
   S703_LM_DC_1ST_CLAMP2.Error_T2.ET := T#0MS;
   S703_LM_DC_1ST_CLAMP2.Error_T2.STATE := B#16#0;
   S703_LM_DC_1ST_CLAMP2.Error_T2.STIME := T#0MS;
   S703_LM_DC_1ST_CLAMP2.Error_T2.ATIME := T#0MS;
   S703_LM_DC_1ST_CLAMP2.CHK_Aux1 := FALSE;
   S703_LM_DC_1ST_CLAMP2.CHK_Aux2 := FALSE;
   S703_LM_DC_1ST_CLAMP2.Error_T1_DN := FALSE;
   S703_LM_DC_1ST_CLAMP2.Error_T2_DN := FALSE;
   S703_LM_DC_1ST_CLAMP2.Adv_Memo := FALSE;
   S703_LM_DC_1ST_CLAMP2.Visu_Adv_Arr[0] := FALSE;
   S703_LM_DC_1ST_CLAMP2.Visu_Adv_Arr[1] := FALSE;
   S703_LM_DC_1ST_CLAMP2.Visu_Adv_Arr[2] := FALSE;
   S703_LM_DC_1ST_CLAMP2.Visu_Adv_Arr[3] := FALSE;
   S703_LM_DC_1ST_CLAMP2.Visu_Adv_Arr[4] := FALSE;
   S703_LM_DC_1ST_CLAMP2.Visu_Adv_Arr[5] := FALSE;
   S703_LM_DC_1ST_CLAMP2.Visu_Adv_Arr[6] := FALSE;
   S703_LM_DC_1ST_CLAMP2.Visu_Adv_Arr[7] := FALSE;
   S703_LM_DC_1ST_CLAMP2.Visu_Adv_Arr[8] := FALSE;
   S703_LM_DC_1ST_CLAMP2.Visu_Adv_Arr[9] := FALSE;
   S703_LM_DC_1ST_CLAMP2.Visu_Adv_Arr[10] := FALSE;
   S703_LM_DC_1ST_CLAMP2.Visu_Adv_Arr[11] := FALSE;
   S703_LM_DC_1ST_CLAMP2.Visu_Adv_Arr[12] := FALSE;
   S703_LM_DC_1ST_CLAMP2.Visu_Adv_Arr[13] := FALSE;
   S703_LM_DC_1ST_CLAMP2.Visu_Adv_Arr[14] := FALSE;
   S703_LM_DC_1ST_CLAMP2.Visu_Adv_Arr[15] := FALSE;
   S703_LM_DC_1ST_CLAMP2.Visu_Ret_Arr[0] := FALSE;
   S703_LM_DC_1ST_CLAMP2.Visu_Ret_Arr[1] := FALSE;
   S703_LM_DC_1ST_CLAMP2.Visu_Ret_Arr[2] := FALSE;
   S703_LM_DC_1ST_CLAMP2.Visu_Ret_Arr[3] := FALSE;
   S703_LM_DC_1ST_CLAMP2.Visu_Ret_Arr[4] := FALSE;
   S703_LM_DC_1ST_CLAMP2.Visu_Ret_Arr[5] := FALSE;
   S703_LM_DC_1ST_CLAMP2.Visu_Ret_Arr[6] := FALSE;
   S703_LM_DC_1ST_CLAMP2.Visu_Ret_Arr[7] := FALSE;
   S703_LM_DC_1ST_CLAMP2.Visu_Ret_Arr[8] := FALSE;
   S703_LM_DC_1ST_CLAMP2.Visu_Ret_Arr[9] := FALSE;
   S703_LM_DC_1ST_CLAMP2.Visu_Ret_Arr[10] := FALSE;
   S703_LM_DC_1ST_CLAMP2.Visu_Ret_Arr[11] := FALSE;
   S703_LM_DC_1ST_CLAMP2.Visu_Ret_Arr[12] := FALSE;
   S703_LM_DC_1ST_CLAMP2.Visu_Ret_Arr[13] := FALSE;
   S703_LM_DC_1ST_CLAMP2.Visu_Ret_Arr[14] := FALSE;
   S703_LM_DC_1ST_CLAMP2.Visu_Ret_Arr[15] := FALSE;
   S703_LM_DC_1ST_CLAMP2.BLK_Move_Ret := 0;
   S703_LM_DC_1ST_CLAMP2.Enable := FALSE;
   S703_LM_DC_1ST_CLAMP2.Adv_End := FALSE;
   S703_LM_DC_1ST_CLAMP2.Ret_End := FALSE;
   S703_LM_DC_1ST_CLAMP3.Enable_Aux := FALSE;
   S703_LM_DC_1ST_CLAMP3.Adv_Amount := 0;
   S703_LM_DC_1ST_CLAMP3.Ret_Amount := 0;
   S703_LM_DC_1ST_CLAMP3.LS_Adv1 := FALSE;
   S703_LM_DC_1ST_CLAMP3.LS_Ret1 := FALSE;
   S703_LM_DC_1ST_CLAMP3.LS_Adv2 := FALSE;
   S703_LM_DC_1ST_CLAMP3.LS_Ret2 := FALSE;
   S703_LM_DC_1ST_CLAMP3.LS_Adv3 := FALSE;
   S703_LM_DC_1ST_CLAMP3.LS_Ret3 := FALSE;
   S703_LM_DC_1ST_CLAMP3.LS_Adv4 := FALSE;
   S703_LM_DC_1ST_CLAMP3.LS_Ret4 := FALSE;
   S703_LM_DC_1ST_CLAMP3.SOL_Adv := FALSE;
   S703_LM_DC_1ST_CLAMP3.SOL_Ret := FALSE;
   S703_LM_DC_1ST_CLAMP3.M_Ready := FALSE;
   S703_LM_DC_1ST_CLAMP3.T_CHK1 := T#0MS;
   S703_LM_DC_1ST_CLAMP3.T_CHK2 := T#0MS;
   S703_LM_DC_1ST_CLAMP3.PB_Lamp_CHK := FALSE;
   S703_LM_DC_1ST_CLAMP3.PB_Error_Rst := FALSE;
   S703_LM_DC_1ST_CLAMP3.M_FLICK := FALSE;
   S703_LM_DC_1ST_CLAMP3.M_Adv_Err := FALSE;
   S703_LM_DC_1ST_CLAMP3.M_Ret_Err := FALSE;
   S703_LM_DC_1ST_CLAMP3.LP_Adv := FALSE;
   S703_LM_DC_1ST_CLAMP3.LP_Ret := FALSE;
   S703_LM_DC_1ST_CLAMP3.Visu_Adv := W#16#0;
   S703_LM_DC_1ST_CLAMP3.Visu_Ret := W#16#0;
   S703_LM_DC_1ST_CLAMP3.Error_T1.IN := FALSE;
   S703_LM_DC_1ST_CLAMP3.Error_T1.PT := T#0MS;
   S703_LM_DC_1ST_CLAMP3.Error_T1.Q := FALSE;
   S703_LM_DC_1ST_CLAMP3.Error_T1.ET := T#0MS;
   S703_LM_DC_1ST_CLAMP3.Error_T1.STATE := B#16#0;
   S703_LM_DC_1ST_CLAMP3.Error_T1.STIME := T#0MS;
   S703_LM_DC_1ST_CLAMP3.Error_T1.ATIME := T#0MS;
   S703_LM_DC_1ST_CLAMP3.Error_T2.IN := FALSE;
   S703_LM_DC_1ST_CLAMP3.Error_T2.PT := T#0MS;
   S703_LM_DC_1ST_CLAMP3.Error_T2.Q := FALSE;
   S703_LM_DC_1ST_CLAMP3.Error_T2.ET := T#0MS;
   S703_LM_DC_1ST_CLAMP3.Error_T2.STATE := B#16#0;
   S703_LM_DC_1ST_CLAMP3.Error_T2.STIME := T#0MS;
   S703_LM_DC_1ST_CLAMP3.Error_T2.ATIME := T#0MS;
   S703_LM_DC_1ST_CLAMP3.CHK_Aux1 := FALSE;
   S703_LM_DC_1ST_CLAMP3.CHK_Aux2 := FALSE;
   S703_LM_DC_1ST_CLAMP3.Error_T1_DN := FALSE;
   S703_LM_DC_1ST_CLAMP3.Error_T2_DN := FALSE;
   S703_LM_DC_1ST_CLAMP3.Adv_Memo := FALSE;
   S703_LM_DC_1ST_CLAMP3.Visu_Adv_Arr[0] := FALSE;
   S703_LM_DC_1ST_CLAMP3.Visu_Adv_Arr[1] := FALSE;
   S703_LM_DC_1ST_CLAMP3.Visu_Adv_Arr[2] := FALSE;
   S703_LM_DC_1ST_CLAMP3.Visu_Adv_Arr[3] := FALSE;
   S703_LM_DC_1ST_CLAMP3.Visu_Adv_Arr[4] := FALSE;
   S703_LM_DC_1ST_CLAMP3.Visu_Adv_Arr[5] := FALSE;
   S703_LM_DC_1ST_CLAMP3.Visu_Adv_Arr[6] := FALSE;
   S703_LM_DC_1ST_CLAMP3.Visu_Adv_Arr[7] := FALSE;
   S703_LM_DC_1ST_CLAMP3.Visu_Adv_Arr[8] := FALSE;
   S703_LM_DC_1ST_CLAMP3.Visu_Adv_Arr[9] := FALSE;
   S703_LM_DC_1ST_CLAMP3.Visu_Adv_Arr[10] := FALSE;
   S703_LM_DC_1ST_CLAMP3.Visu_Adv_Arr[11] := FALSE;
   S703_LM_DC_1ST_CLAMP3.Visu_Adv_Arr[12] := FALSE;
   S703_LM_DC_1ST_CLAMP3.Visu_Adv_Arr[13] := FALSE;
   S703_LM_DC_1ST_CLAMP3.Visu_Adv_Arr[14] := FALSE;
   S703_LM_DC_1ST_CLAMP3.Visu_Adv_Arr[15] := FALSE;
   S703_LM_DC_1ST_CLAMP3.Visu_Ret_Arr[0] := FALSE;
   S703_LM_DC_1ST_CLAMP3.Visu_Ret_Arr[1] := FALSE;
   S703_LM_DC_1ST_CLAMP3.Visu_Ret_Arr[2] := FALSE;
   S703_LM_DC_1ST_CLAMP3.Visu_Ret_Arr[3] := FALSE;
   S703_LM_DC_1ST_CLAMP3.Visu_Ret_Arr[4] := FALSE;
   S703_LM_DC_1ST_CLAMP3.Visu_Ret_Arr[5] := FALSE;
   S703_LM_DC_1ST_CLAMP3.Visu_Ret_Arr[6] := FALSE;
   S703_LM_DC_1ST_CLAMP3.Visu_Ret_Arr[7] := FALSE;
   S703_LM_DC_1ST_CLAMP3.Visu_Ret_Arr[8] := FALSE;
   S703_LM_DC_1ST_CLAMP3.Visu_Ret_Arr[9] := FALSE;
   S703_LM_DC_1ST_CLAMP3.Visu_Ret_Arr[10] := FALSE;
   S703_LM_DC_1ST_CLAMP3.Visu_Ret_Arr[11] := FALSE;
   S703_LM_DC_1ST_CLAMP3.Visu_Ret_Arr[12] := FALSE;
   S703_LM_DC_1ST_CLAMP3.Visu_Ret_Arr[13] := FALSE;
   S703_LM_DC_1ST_CLAMP3.Visu_Ret_Arr[14] := FALSE;
   S703_LM_DC_1ST_CLAMP3.Visu_Ret_Arr[15] := FALSE;
   S703_LM_DC_1ST_CLAMP3.BLK_Move_Ret := 0;
   S703_LM_DC_1ST_CLAMP3.Enable := FALSE;
   S703_LM_DC_1ST_CLAMP3.Adv_End := FALSE;
   S703_LM_DC_1ST_CLAMP3.Ret_End := FALSE;
   S703_LM_DC_1ST_CLAMP4.Enable_Aux := FALSE;
   S703_LM_DC_1ST_CLAMP4.Adv_Amount := 0;
   S703_LM_DC_1ST_CLAMP4.Ret_Amount := 0;
   S703_LM_DC_1ST_CLAMP4.LS_Adv1 := FALSE;
   S703_LM_DC_1ST_CLAMP4.LS_Ret1 := FALSE;
   S703_LM_DC_1ST_CLAMP4.LS_Adv2 := FALSE;
   S703_LM_DC_1ST_CLAMP4.LS_Ret2 := FALSE;
   S703_LM_DC_1ST_CLAMP4.LS_Adv3 := FALSE;
   S703_LM_DC_1ST_CLAMP4.LS_Ret3 := FALSE;
   S703_LM_DC_1ST_CLAMP4.LS_Adv4 := FALSE;
   S703_LM_DC_1ST_CLAMP4.LS_Ret4 := FALSE;
   S703_LM_DC_1ST_CLAMP4.SOL_Adv := FALSE;
   S703_LM_DC_1ST_CLAMP4.SOL_Ret := FALSE;
   S703_LM_DC_1ST_CLAMP4.M_Ready := FALSE;
   S703_LM_DC_1ST_CLAMP4.T_CHK1 := T#0MS;
   S703_LM_DC_1ST_CLAMP4.T_CHK2 := T#0MS;
   S703_LM_DC_1ST_CLAMP4.PB_Lamp_CHK := FALSE;
   S703_LM_DC_1ST_CLAMP4.PB_Error_Rst := FALSE;
   S703_LM_DC_1ST_CLAMP4.M_FLICK := FALSE;
   S703_LM_DC_1ST_CLAMP4.M_Adv_Err := FALSE;
   S703_LM_DC_1ST_CLAMP4.M_Ret_Err := FALSE;
   S703_LM_DC_1ST_CLAMP4.LP_Adv := FALSE;
   S703_LM_DC_1ST_CLAMP4.LP_Ret := FALSE;
   S703_LM_DC_1ST_CLAMP4.Visu_Adv := W#16#0;
   S703_LM_DC_1ST_CLAMP4.Visu_Ret := W#16#0;
   S703_LM_DC_1ST_CLAMP4.Error_T1.IN := FALSE;
   S703_LM_DC_1ST_CLAMP4.Error_T1.PT := T#0MS;
   S703_LM_DC_1ST_CLAMP4.Error_T1.Q := FALSE;
   S703_LM_DC_1ST_CLAMP4.Error_T1.ET := T#0MS;
   S703_LM_DC_1ST_CLAMP4.Error_T1.STATE := B#16#0;
   S703_LM_DC_1ST_CLAMP4.Error_T1.STIME := T#0MS;
   S703_LM_DC_1ST_CLAMP4.Error_T1.ATIME := T#0MS;
   S703_LM_DC_1ST_CLAMP4.Error_T2.IN := FALSE;
   S703_LM_DC_1ST_CLAMP4.Error_T2.PT := T#0MS;
   S703_LM_DC_1ST_CLAMP4.Error_T2.Q := FALSE;
   S703_LM_DC_1ST_CLAMP4.Error_T2.ET := T#0MS;
   S703_LM_DC_1ST_CLAMP4.Error_T2.STATE := B#16#0;
   S703_LM_DC_1ST_CLAMP4.Error_T2.STIME := T#0MS;
   S703_LM_DC_1ST_CLAMP4.Error_T2.ATIME := T#0MS;
   S703_LM_DC_1ST_CLAMP4.CHK_Aux1 := FALSE;
   S703_LM_DC_1ST_CLAMP4.CHK_Aux2 := FALSE;
   S703_LM_DC_1ST_CLAMP4.Error_T1_DN := FALSE;
   S703_LM_DC_1ST_CLAMP4.Error_T2_DN := FALSE;
   S703_LM_DC_1ST_CLAMP4.Adv_Memo := FALSE;
   S703_LM_DC_1ST_CLAMP4.Visu_Adv_Arr[0] := FALSE;
   S703_LM_DC_1ST_CLAMP4.Visu_Adv_Arr[1] := FALSE;
   S703_LM_DC_1ST_CLAMP4.Visu_Adv_Arr[2] := FALSE;
   S703_LM_DC_1ST_CLAMP4.Visu_Adv_Arr[3] := FALSE;
   S703_LM_DC_1ST_CLAMP4.Visu_Adv_Arr[4] := FALSE;
   S703_LM_DC_1ST_CLAMP4.Visu_Adv_Arr[5] := FALSE;
   S703_LM_DC_1ST_CLAMP4.Visu_Adv_Arr[6] := FALSE;
   S703_LM_DC_1ST_CLAMP4.Visu_Adv_Arr[7] := FALSE;
   S703_LM_DC_1ST_CLAMP4.Visu_Adv_Arr[8] := FALSE;
   S703_LM_DC_1ST_CLAMP4.Visu_Adv_Arr[9] := FALSE;
   S703_LM_DC_1ST_CLAMP4.Visu_Adv_Arr[10] := FALSE;
   S703_LM_DC_1ST_CLAMP4.Visu_Adv_Arr[11] := FALSE;
   S703_LM_DC_1ST_CLAMP4.Visu_Adv_Arr[12] := FALSE;
   S703_LM_DC_1ST_CLAMP4.Visu_Adv_Arr[13] := FALSE;
   S703_LM_DC_1ST_CLAMP4.Visu_Adv_Arr[14] := FALSE;
   S703_LM_DC_1ST_CLAMP4.Visu_Adv_Arr[15] := FALSE;
   S703_LM_DC_1ST_CLAMP4.Visu_Ret_Arr[0] := FALSE;
   S703_LM_DC_1ST_CLAMP4.Visu_Ret_Arr[1] := FALSE;
   S703_LM_DC_1ST_CLAMP4.Visu_Ret_Arr[2] := FALSE;
   S703_LM_DC_1ST_CLAMP4.Visu_Ret_Arr[3] := FALSE;
   S703_LM_DC_1ST_CLAMP4.Visu_Ret_Arr[4] := FALSE;
   S703_LM_DC_1ST_CLAMP4.Visu_Ret_Arr[5] := FALSE;
   S703_LM_DC_1ST_CLAMP4.Visu_Ret_Arr[6] := FALSE;
   S703_LM_DC_1ST_CLAMP4.Visu_Ret_Arr[7] := FALSE;
   S703_LM_DC_1ST_CLAMP4.Visu_Ret_Arr[8] := FALSE;
   S703_LM_DC_1ST_CLAMP4.Visu_Ret_Arr[9] := FALSE;
   S703_LM_DC_1ST_CLAMP4.Visu_Ret_Arr[10] := FALSE;
   S703_LM_DC_1ST_CLAMP4.Visu_Ret_Arr[11] := FALSE;
   S703_LM_DC_1ST_CLAMP4.Visu_Ret_Arr[12] := FALSE;
   S703_LM_DC_1ST_CLAMP4.Visu_Ret_Arr[13] := FALSE;
   S703_LM_DC_1ST_CLAMP4.Visu_Ret_Arr[14] := FALSE;
   S703_LM_DC_1ST_CLAMP4.Visu_Ret_Arr[15] := FALSE;
   S703_LM_DC_1ST_CLAMP4.BLK_Move_Ret := 0;
   S703_LM_DC_1ST_CLAMP4.Enable := FALSE;
   S703_LM_DC_1ST_CLAMP4.Adv_End := FALSE;
   S703_LM_DC_1ST_CLAMP4.Ret_End := FALSE;
   S703_LM_DC_2ND_CLAMP1.Enable_Aux := FALSE;
   S703_LM_DC_2ND_CLAMP1.Adv_Amount := 0;
   S703_LM_DC_2ND_CLAMP1.Ret_Amount := 0;
   S703_LM_DC_2ND_CLAMP1.LS_Adv1 := FALSE;
   S703_LM_DC_2ND_CLAMP1.LS_Ret1 := FALSE;
   S703_LM_DC_2ND_CLAMP1.LS_Adv2 := FALSE;
   S703_LM_DC_2ND_CLAMP1.LS_Ret2 := FALSE;
   S703_LM_DC_2ND_CLAMP1.LS_Adv3 := FALSE;
   S703_LM_DC_2ND_CLAMP1.LS_Ret3 := FALSE;
   S703_LM_DC_2ND_CLAMP1.LS_Adv4 := FALSE;
   S703_LM_DC_2ND_CLAMP1.LS_Ret4 := FALSE;
   S703_LM_DC_2ND_CLAMP1.SOL_Adv := FALSE;
   S703_LM_DC_2ND_CLAMP1.SOL_Ret := FALSE;
   S703_LM_DC_2ND_CLAMP1.M_Ready := FALSE;
   S703_LM_DC_2ND_CLAMP1.T_CHK1 := T#0MS;
   S703_LM_DC_2ND_CLAMP1.T_CHK2 := T#0MS;
   S703_LM_DC_2ND_CLAMP1.PB_Lamp_CHK := FALSE;
   S703_LM_DC_2ND_CLAMP1.PB_Error_Rst := FALSE;
   S703_LM_DC_2ND_CLAMP1.M_FLICK := FALSE;
   S703_LM_DC_2ND_CLAMP1.M_Adv_Err := FALSE;
   S703_LM_DC_2ND_CLAMP1.M_Ret_Err := FALSE;
   S703_LM_DC_2ND_CLAMP1.LP_Adv := FALSE;
   S703_LM_DC_2ND_CLAMP1.LP_Ret := FALSE;
   S703_LM_DC_2ND_CLAMP1.Visu_Adv := W#16#0;
   S703_LM_DC_2ND_CLAMP1.Visu_Ret := W#16#0;
   S703_LM_DC_2ND_CLAMP1.Error_T1.IN := FALSE;
   S703_LM_DC_2ND_CLAMP1.Error_T1.PT := T#0MS;
   S703_LM_DC_2ND_CLAMP1.Error_T1.Q := FALSE;
   S703_LM_DC_2ND_CLAMP1.Error_T1.ET := T#0MS;
   S703_LM_DC_2ND_CLAMP1.Error_T1.STATE := B#16#0;
   S703_LM_DC_2ND_CLAMP1.Error_T1.STIME := T#0MS;
   S703_LM_DC_2ND_CLAMP1.Error_T1.ATIME := T#0MS;
   S703_LM_DC_2ND_CLAMP1.Error_T2.IN := FALSE;
   S703_LM_DC_2ND_CLAMP1.Error_T2.PT := T#0MS;
   S703_LM_DC_2ND_CLAMP1.Error_T2.Q := FALSE;
   S703_LM_DC_2ND_CLAMP1.Error_T2.ET := T#0MS;
   S703_LM_DC_2ND_CLAMP1.Error_T2.STATE := B#16#0;
   S703_LM_DC_2ND_CLAMP1.Error_T2.STIME := T#0MS;
   S703_LM_DC_2ND_CLAMP1.Error_T2.ATIME := T#0MS;
   S703_LM_DC_2ND_CLAMP1.CHK_Aux1 := FALSE;
   S703_LM_DC_2ND_CLAMP1.CHK_Aux2 := FALSE;
   S703_LM_DC_2ND_CLAMP1.Error_T1_DN := FALSE;
   S703_LM_DC_2ND_CLAMP1.Error_T2_DN := FALSE;
   S703_LM_DC_2ND_CLAMP1.Adv_Memo := FALSE;
   S703_LM_DC_2ND_CLAMP1.Visu_Adv_Arr[0] := FALSE;
   S703_LM_DC_2ND_CLAMP1.Visu_Adv_Arr[1] := FALSE;
   S703_LM_DC_2ND_CLAMP1.Visu_Adv_Arr[2] := FALSE;
   S703_LM_DC_2ND_CLAMP1.Visu_Adv_Arr[3] := FALSE;
   S703_LM_DC_2ND_CLAMP1.Visu_Adv_Arr[4] := FALSE;
   S703_LM_DC_2ND_CLAMP1.Visu_Adv_Arr[5] := FALSE;
   S703_LM_DC_2ND_CLAMP1.Visu_Adv_Arr[6] := FALSE;
   S703_LM_DC_2ND_CLAMP1.Visu_Adv_Arr[7] := FALSE;
   S703_LM_DC_2ND_CLAMP1.Visu_Adv_Arr[8] := FALSE;
   S703_LM_DC_2ND_CLAMP1.Visu_Adv_Arr[9] := FALSE;
   S703_LM_DC_2ND_CLAMP1.Visu_Adv_Arr[10] := FALSE;
   S703_LM_DC_2ND_CLAMP1.Visu_Adv_Arr[11] := FALSE;
   S703_LM_DC_2ND_CLAMP1.Visu_Adv_Arr[12] := FALSE;
   S703_LM_DC_2ND_CLAMP1.Visu_Adv_Arr[13] := FALSE;
   S703_LM_DC_2ND_CLAMP1.Visu_Adv_Arr[14] := FALSE;
   S703_LM_DC_2ND_CLAMP1.Visu_Adv_Arr[15] := FALSE;
   S703_LM_DC_2ND_CLAMP1.Visu_Ret_Arr[0] := FALSE;
   S703_LM_DC_2ND_CLAMP1.Visu_Ret_Arr[1] := FALSE;
   S703_LM_DC_2ND_CLAMP1.Visu_Ret_Arr[2] := FALSE;
   S703_LM_DC_2ND_CLAMP1.Visu_Ret_Arr[3] := FALSE;
   S703_LM_DC_2ND_CLAMP1.Visu_Ret_Arr[4] := FALSE;
   S703_LM_DC_2ND_CLAMP1.Visu_Ret_Arr[5] := FALSE;
   S703_LM_DC_2ND_CLAMP1.Visu_Ret_Arr[6] := FALSE;
   S703_LM_DC_2ND_CLAMP1.Visu_Ret_Arr[7] := FALSE;
   S703_LM_DC_2ND_CLAMP1.Visu_Ret_Arr[8] := FALSE;
   S703_LM_DC_2ND_CLAMP1.Visu_Ret_Arr[9] := FALSE;
   S703_LM_DC_2ND_CLAMP1.Visu_Ret_Arr[10] := FALSE;
   S703_LM_DC_2ND_CLAMP1.Visu_Ret_Arr[11] := FALSE;
   S703_LM_DC_2ND_CLAMP1.Visu_Ret_Arr[12] := FALSE;
   S703_LM_DC_2ND_CLAMP1.Visu_Ret_Arr[13] := FALSE;
   S703_LM_DC_2ND_CLAMP1.Visu_Ret_Arr[14] := FALSE;
   S703_LM_DC_2ND_CLAMP1.Visu_Ret_Arr[15] := FALSE;
   S703_LM_DC_2ND_CLAMP1.BLK_Move_Ret := 0;
   S703_LM_DC_2ND_CLAMP1.Enable := FALSE;
   S703_LM_DC_2ND_CLAMP1.Adv_End := FALSE;
   S703_LM_DC_2ND_CLAMP1.Ret_End := FALSE;
   S703_LM_DC_2ND_CLAMP2.Enable_Aux := FALSE;
   S703_LM_DC_2ND_CLAMP2.Adv_Amount := 0;
   S703_LM_DC_2ND_CLAMP2.Ret_Amount := 0;
   S703_LM_DC_2ND_CLAMP2.LS_Adv1 := FALSE;
   S703_LM_DC_2ND_CLAMP2.LS_Ret1 := FALSE;
   S703_LM_DC_2ND_CLAMP2.LS_Adv2 := FALSE;
   S703_LM_DC_2ND_CLAMP2.LS_Ret2 := FALSE;
   S703_LM_DC_2ND_CLAMP2.LS_Adv3 := FALSE;
   S703_LM_DC_2ND_CLAMP2.LS_Ret3 := FALSE;
   S703_LM_DC_2ND_CLAMP2.LS_Adv4 := FALSE;
   S703_LM_DC_2ND_CLAMP2.LS_Ret4 := FALSE;
   S703_LM_DC_2ND_CLAMP2.SOL_Adv := FALSE;
   S703_LM_DC_2ND_CLAMP2.SOL_Ret := FALSE;
   S703_LM_DC_2ND_CLAMP2.M_Ready := FALSE;
   S703_LM_DC_2ND_CLAMP2.T_CHK1 := T#0MS;
   S703_LM_DC_2ND_CLAMP2.T_CHK2 := T#0MS;
   S703_LM_DC_2ND_CLAMP2.PB_Lamp_CHK := FALSE;
   S703_LM_DC_2ND_CLAMP2.PB_Error_Rst := FALSE;
   S703_LM_DC_2ND_CLAMP2.M_FLICK := FALSE;
   S703_LM_DC_2ND_CLAMP2.M_Adv_Err := FALSE;
   S703_LM_DC_2ND_CLAMP2.M_Ret_Err := FALSE;
   S703_LM_DC_2ND_CLAMP2.LP_Adv := FALSE;
   S703_LM_DC_2ND_CLAMP2.LP_Ret := FALSE;
   S703_LM_DC_2ND_CLAMP2.Visu_Adv := W#16#0;
   S703_LM_DC_2ND_CLAMP2.Visu_Ret := W#16#0;
   S703_LM_DC_2ND_CLAMP2.Error_T1.IN := FALSE;
   S703_LM_DC_2ND_CLAMP2.Error_T1.PT := T#0MS;
   S703_LM_DC_2ND_CLAMP2.Error_T1.Q := FALSE;
   S703_LM_DC_2ND_CLAMP2.Error_T1.ET := T#0MS;
   S703_LM_DC_2ND_CLAMP2.Error_T1.STATE := B#16#0;
   S703_LM_DC_2ND_CLAMP2.Error_T1.STIME := T#0MS;
   S703_LM_DC_2ND_CLAMP2.Error_T1.ATIME := T#0MS;
   S703_LM_DC_2ND_CLAMP2.Error_T2.IN := FALSE;
   S703_LM_DC_2ND_CLAMP2.Error_T2.PT := T#0MS;
   S703_LM_DC_2ND_CLAMP2.Error_T2.Q := FALSE;
   S703_LM_DC_2ND_CLAMP2.Error_T2.ET := T#0MS;
   S703_LM_DC_2ND_CLAMP2.Error_T2.STATE := B#16#0;
   S703_LM_DC_2ND_CLAMP2.Error_T2.STIME := T#0MS;
   S703_LM_DC_2ND_CLAMP2.Error_T2.ATIME := T#0MS;
   S703_LM_DC_2ND_CLAMP2.CHK_Aux1 := FALSE;
   S703_LM_DC_2ND_CLAMP2.CHK_Aux2 := FALSE;
   S703_LM_DC_2ND_CLAMP2.Error_T1_DN := FALSE;
   S703_LM_DC_2ND_CLAMP2.Error_T2_DN := FALSE;
   S703_LM_DC_2ND_CLAMP2.Adv_Memo := FALSE;
   S703_LM_DC_2ND_CLAMP2.Visu_Adv_Arr[0] := FALSE;
   S703_LM_DC_2ND_CLAMP2.Visu_Adv_Arr[1] := FALSE;
   S703_LM_DC_2ND_CLAMP2.Visu_Adv_Arr[2] := FALSE;
   S703_LM_DC_2ND_CLAMP2.Visu_Adv_Arr[3] := FALSE;
   S703_LM_DC_2ND_CLAMP2.Visu_Adv_Arr[4] := FALSE;
   S703_LM_DC_2ND_CLAMP2.Visu_Adv_Arr[5] := FALSE;
   S703_LM_DC_2ND_CLAMP2.Visu_Adv_Arr[6] := FALSE;
   S703_LM_DC_2ND_CLAMP2.Visu_Adv_Arr[7] := FALSE;
   S703_LM_DC_2ND_CLAMP2.Visu_Adv_Arr[8] := FALSE;
   S703_LM_DC_2ND_CLAMP2.Visu_Adv_Arr[9] := FALSE;
   S703_LM_DC_2ND_CLAMP2.Visu_Adv_Arr[10] := FALSE;
   S703_LM_DC_2ND_CLAMP2.Visu_Adv_Arr[11] := FALSE;
   S703_LM_DC_2ND_CLAMP2.Visu_Adv_Arr[12] := FALSE;
   S703_LM_DC_2ND_CLAMP2.Visu_Adv_Arr[13] := FALSE;
   S703_LM_DC_2ND_CLAMP2.Visu_Adv_Arr[14] := FALSE;
   S703_LM_DC_2ND_CLAMP2.Visu_Adv_Arr[15] := FALSE;
   S703_LM_DC_2ND_CLAMP2.Visu_Ret_Arr[0] := FALSE;
   S703_LM_DC_2ND_CLAMP2.Visu_Ret_Arr[1] := FALSE;
   S703_LM_DC_2ND_CLAMP2.Visu_Ret_Arr[2] := FALSE;
   S703_LM_DC_2ND_CLAMP2.Visu_Ret_Arr[3] := FALSE;
   S703_LM_DC_2ND_CLAMP2.Visu_Ret_Arr[4] := FALSE;
   S703_LM_DC_2ND_CLAMP2.Visu_Ret_Arr[5] := FALSE;
   S703_LM_DC_2ND_CLAMP2.Visu_Ret_Arr[6] := FALSE;
   S703_LM_DC_2ND_CLAMP2.Visu_Ret_Arr[7] := FALSE;
   S703_LM_DC_2ND_CLAMP2.Visu_Ret_Arr[8] := FALSE;
   S703_LM_DC_2ND_CLAMP2.Visu_Ret_Arr[9] := FALSE;
   S703_LM_DC_2ND_CLAMP2.Visu_Ret_Arr[10] := FALSE;
   S703_LM_DC_2ND_CLAMP2.Visu_Ret_Arr[11] := FALSE;
   S703_LM_DC_2ND_CLAMP2.Visu_Ret_Arr[12] := FALSE;
   S703_LM_DC_2ND_CLAMP2.Visu_Ret_Arr[13] := FALSE;
   S703_LM_DC_2ND_CLAMP2.Visu_Ret_Arr[14] := FALSE;
   S703_LM_DC_2ND_CLAMP2.Visu_Ret_Arr[15] := FALSE;
   S703_LM_DC_2ND_CLAMP2.BLK_Move_Ret := 0;
   S703_LM_DC_2ND_CLAMP2.Enable := FALSE;
   S703_LM_DC_2ND_CLAMP2.Adv_End := FALSE;
   S703_LM_DC_2ND_CLAMP2.Ret_End := FALSE;
   S703_LM_DC_2ND_CLAMP3.Enable_Aux := FALSE;
   S703_LM_DC_2ND_CLAMP3.Adv_Amount := 0;
   S703_LM_DC_2ND_CLAMP3.Ret_Amount := 0;
   S703_LM_DC_2ND_CLAMP3.LS_Adv1 := FALSE;
   S703_LM_DC_2ND_CLAMP3.LS_Ret1 := FALSE;
   S703_LM_DC_2ND_CLAMP3.LS_Adv2 := FALSE;
   S703_LM_DC_2ND_CLAMP3.LS_Ret2 := FALSE;
   S703_LM_DC_2ND_CLAMP3.LS_Adv3 := FALSE;
   S703_LM_DC_2ND_CLAMP3.LS_Ret3 := FALSE;
   S703_LM_DC_2ND_CLAMP3.LS_Adv4 := FALSE;
   S703_LM_DC_2ND_CLAMP3.LS_Ret4 := FALSE;
   S703_LM_DC_2ND_CLAMP3.SOL_Adv := FALSE;
   S703_LM_DC_2ND_CLAMP3.SOL_Ret := FALSE;
   S703_LM_DC_2ND_CLAMP3.M_Ready := FALSE;
   S703_LM_DC_2ND_CLAMP3.T_CHK1 := T#0MS;
   S703_LM_DC_2ND_CLAMP3.T_CHK2 := T#0MS;
   S703_LM_DC_2ND_CLAMP3.PB_Lamp_CHK := FALSE;
   S703_LM_DC_2ND_CLAMP3.PB_Error_Rst := FALSE;
   S703_LM_DC_2ND_CLAMP3.M_FLICK := FALSE;
   S703_LM_DC_2ND_CLAMP3.M_Adv_Err := FALSE;
   S703_LM_DC_2ND_CLAMP3.M_Ret_Err := FALSE;
   S703_LM_DC_2ND_CLAMP3.LP_Adv := FALSE;
   S703_LM_DC_2ND_CLAMP3.LP_Ret := FALSE;
   S703_LM_DC_2ND_CLAMP3.Visu_Adv := W#16#0;
   S703_LM_DC_2ND_CLAMP3.Visu_Ret := W#16#0;
   S703_LM_DC_2ND_CLAMP3.Error_T1.IN := FALSE;
   S703_LM_DC_2ND_CLAMP3.Error_T1.PT := T#0MS;
   S703_LM_DC_2ND_CLAMP3.Error_T1.Q := FALSE;
   S703_LM_DC_2ND_CLAMP3.Error_T1.ET := T#0MS;
   S703_LM_DC_2ND_CLAMP3.Error_T1.STATE := B#16#0;
   S703_LM_DC_2ND_CLAMP3.Error_T1.STIME := T#0MS;
   S703_LM_DC_2ND_CLAMP3.Error_T1.ATIME := T#0MS;
   S703_LM_DC_2ND_CLAMP3.Error_T2.IN := FALSE;
   S703_LM_DC_2ND_CLAMP3.Error_T2.PT := T#0MS;
   S703_LM_DC_2ND_CLAMP3.Error_T2.Q := FALSE;
   S703_LM_DC_2ND_CLAMP3.Error_T2.ET := T#0MS;
   S703_LM_DC_2ND_CLAMP3.Error_T2.STATE := B#16#0;
   S703_LM_DC_2ND_CLAMP3.Error_T2.STIME := T#0MS;
   S703_LM_DC_2ND_CLAMP3.Error_T2.ATIME := T#0MS;
   S703_LM_DC_2ND_CLAMP3.CHK_Aux1 := FALSE;
   S703_LM_DC_2ND_CLAMP3.CHK_Aux2 := FALSE;
   S703_LM_DC_2ND_CLAMP3.Error_T1_DN := FALSE;
   S703_LM_DC_2ND_CLAMP3.Error_T2_DN := FALSE;
   S703_LM_DC_2ND_CLAMP3.Adv_Memo := FALSE;
   S703_LM_DC_2ND_CLAMP3.Visu_Adv_Arr[0] := FALSE;
   S703_LM_DC_2ND_CLAMP3.Visu_Adv_Arr[1] := FALSE;
   S703_LM_DC_2ND_CLAMP3.Visu_Adv_Arr[2] := FALSE;
   S703_LM_DC_2ND_CLAMP3.Visu_Adv_Arr[3] := FALSE;
   S703_LM_DC_2ND_CLAMP3.Visu_Adv_Arr[4] := FALSE;
   S703_LM_DC_2ND_CLAMP3.Visu_Adv_Arr[5] := FALSE;
   S703_LM_DC_2ND_CLAMP3.Visu_Adv_Arr[6] := FALSE;
   S703_LM_DC_2ND_CLAMP3.Visu_Adv_Arr[7] := FALSE;
   S703_LM_DC_2ND_CLAMP3.Visu_Adv_Arr[8] := FALSE;
   S703_LM_DC_2ND_CLAMP3.Visu_Adv_Arr[9] := FALSE;
   S703_LM_DC_2ND_CLAMP3.Visu_Adv_Arr[10] := FALSE;
   S703_LM_DC_2ND_CLAMP3.Visu_Adv_Arr[11] := FALSE;
   S703_LM_DC_2ND_CLAMP3.Visu_Adv_Arr[12] := FALSE;
   S703_LM_DC_2ND_CLAMP3.Visu_Adv_Arr[13] := FALSE;
   S703_LM_DC_2ND_CLAMP3.Visu_Adv_Arr[14] := FALSE;
   S703_LM_DC_2ND_CLAMP3.Visu_Adv_Arr[15] := FALSE;
   S703_LM_DC_2ND_CLAMP3.Visu_Ret_Arr[0] := FALSE;
   S703_LM_DC_2ND_CLAMP3.Visu_Ret_Arr[1] := FALSE;
   S703_LM_DC_2ND_CLAMP3.Visu_Ret_Arr[2] := FALSE;
   S703_LM_DC_2ND_CLAMP3.Visu_Ret_Arr[3] := FALSE;
   S703_LM_DC_2ND_CLAMP3.Visu_Ret_Arr[4] := FALSE;
   S703_LM_DC_2ND_CLAMP3.Visu_Ret_Arr[5] := FALSE;
   S703_LM_DC_2ND_CLAMP3.Visu_Ret_Arr[6] := FALSE;
   S703_LM_DC_2ND_CLAMP3.Visu_Ret_Arr[7] := FALSE;
   S703_LM_DC_2ND_CLAMP3.Visu_Ret_Arr[8] := FALSE;
   S703_LM_DC_2ND_CLAMP3.Visu_Ret_Arr[9] := FALSE;
   S703_LM_DC_2ND_CLAMP3.Visu_Ret_Arr[10] := FALSE;
   S703_LM_DC_2ND_CLAMP3.Visu_Ret_Arr[11] := FALSE;
   S703_LM_DC_2ND_CLAMP3.Visu_Ret_Arr[12] := FALSE;
   S703_LM_DC_2ND_CLAMP3.Visu_Ret_Arr[13] := FALSE;
   S703_LM_DC_2ND_CLAMP3.Visu_Ret_Arr[14] := FALSE;
   S703_LM_DC_2ND_CLAMP3.Visu_Ret_Arr[15] := FALSE;
   S703_LM_DC_2ND_CLAMP3.BLK_Move_Ret := 0;
   S703_LM_DC_2ND_CLAMP3.Enable := FALSE;
   S703_LM_DC_2ND_CLAMP3.Adv_End := FALSE;
   S703_LM_DC_2ND_CLAMP3.Ret_End := FALSE;
   S703_LM_DC_2ND_CLAMP4.Enable_Aux := FALSE;
   S703_LM_DC_2ND_CLAMP4.Adv_Amount := 0;
   S703_LM_DC_2ND_CLAMP4.Ret_Amount := 0;
   S703_LM_DC_2ND_CLAMP4.LS_Adv1 := FALSE;
   S703_LM_DC_2ND_CLAMP4.LS_Ret1 := FALSE;
   S703_LM_DC_2ND_CLAMP4.LS_Adv2 := FALSE;
   S703_LM_DC_2ND_CLAMP4.LS_Ret2 := FALSE;
   S703_LM_DC_2ND_CLAMP4.LS_Adv3 := FALSE;
   S703_LM_DC_2ND_CLAMP4.LS_Ret3 := FALSE;
   S703_LM_DC_2ND_CLAMP4.LS_Adv4 := FALSE;
   S703_LM_DC_2ND_CLAMP4.LS_Ret4 := FALSE;
   S703_LM_DC_2ND_CLAMP4.SOL_Adv := FALSE;
   S703_LM_DC_2ND_CLAMP4.SOL_Ret := FALSE;
   S703_LM_DC_2ND_CLAMP4.M_Ready := FALSE;
   S703_LM_DC_2ND_CLAMP4.T_CHK1 := T#0MS;
   S703_LM_DC_2ND_CLAMP4.T_CHK2 := T#0MS;
   S703_LM_DC_2ND_CLAMP4.PB_Lamp_CHK := FALSE;
   S703_LM_DC_2ND_CLAMP4.PB_Error_Rst := FALSE;
   S703_LM_DC_2ND_CLAMP4.M_FLICK := FALSE;
   S703_LM_DC_2ND_CLAMP4.M_Adv_Err := FALSE;
   S703_LM_DC_2ND_CLAMP4.M_Ret_Err := FALSE;
   S703_LM_DC_2ND_CLAMP4.LP_Adv := FALSE;
   S703_LM_DC_2ND_CLAMP4.LP_Ret := FALSE;
   S703_LM_DC_2ND_CLAMP4.Visu_Adv := W#16#0;
   S703_LM_DC_2ND_CLAMP4.Visu_Ret := W#16#0;
   S703_LM_DC_2ND_CLAMP4.Error_T1.IN := FALSE;
   S703_LM_DC_2ND_CLAMP4.Error_T1.PT := T#0MS;
   S703_LM_DC_2ND_CLAMP4.Error_T1.Q := FALSE;
   S703_LM_DC_2ND_CLAMP4.Error_T1.ET := T#0MS;
   S703_LM_DC_2ND_CLAMP4.Error_T1.STATE := B#16#0;
   S703_LM_DC_2ND_CLAMP4.Error_T1.STIME := T#0MS;
   S703_LM_DC_2ND_CLAMP4.Error_T1.ATIME := T#0MS;
   S703_LM_DC_2ND_CLAMP4.Error_T2.IN := FALSE;
   S703_LM_DC_2ND_CLAMP4.Error_T2.PT := T#0MS;
   S703_LM_DC_2ND_CLAMP4.Error_T2.Q := FALSE;
   S703_LM_DC_2ND_CLAMP4.Error_T2.ET := T#0MS;
   S703_LM_DC_2ND_CLAMP4.Error_T2.STATE := B#16#0;
   S703_LM_DC_2ND_CLAMP4.Error_T2.STIME := T#0MS;
   S703_LM_DC_2ND_CLAMP4.Error_T2.ATIME := T#0MS;
   S703_LM_DC_2ND_CLAMP4.CHK_Aux1 := FALSE;
   S703_LM_DC_2ND_CLAMP4.CHK_Aux2 := FALSE;
   S703_LM_DC_2ND_CLAMP4.Error_T1_DN := FALSE;
   S703_LM_DC_2ND_CLAMP4.Error_T2_DN := FALSE;
   S703_LM_DC_2ND_CLAMP4.Adv_Memo := FALSE;
   S703_LM_DC_2ND_CLAMP4.Visu_Adv_Arr[0] := FALSE;
   S703_LM_DC_2ND_CLAMP4.Visu_Adv_Arr[1] := FALSE;
   S703_LM_DC_2ND_CLAMP4.Visu_Adv_Arr[2] := FALSE;
   S703_LM_DC_2ND_CLAMP4.Visu_Adv_Arr[3] := FALSE;
   S703_LM_DC_2ND_CLAMP4.Visu_Adv_Arr[4] := FALSE;
   S703_LM_DC_2ND_CLAMP4.Visu_Adv_Arr[5] := FALSE;
   S703_LM_DC_2ND_CLAMP4.Visu_Adv_Arr[6] := FALSE;
   S703_LM_DC_2ND_CLAMP4.Visu_Adv_Arr[7] := FALSE;
   S703_LM_DC_2ND_CLAMP4.Visu_Adv_Arr[8] := FALSE;
   S703_LM_DC_2ND_CLAMP4.Visu_Adv_Arr[9] := FALSE;
   S703_LM_DC_2ND_CLAMP4.Visu_Adv_Arr[10] := FALSE;
   S703_LM_DC_2ND_CLAMP4.Visu_Adv_Arr[11] := FALSE;
   S703_LM_DC_2ND_CLAMP4.Visu_Adv_Arr[12] := FALSE;
   S703_LM_DC_2ND_CLAMP4.Visu_Adv_Arr[13] := FALSE;
   S703_LM_DC_2ND_CLAMP4.Visu_Adv_Arr[14] := FALSE;
   S703_LM_DC_2ND_CLAMP4.Visu_Adv_Arr[15] := FALSE;
   S703_LM_DC_2ND_CLAMP4.Visu_Ret_Arr[0] := FALSE;
   S703_LM_DC_2ND_CLAMP4.Visu_Ret_Arr[1] := FALSE;
   S703_LM_DC_2ND_CLAMP4.Visu_Ret_Arr[2] := FALSE;
   S703_LM_DC_2ND_CLAMP4.Visu_Ret_Arr[3] := FALSE;
   S703_LM_DC_2ND_CLAMP4.Visu_Ret_Arr[4] := FALSE;
   S703_LM_DC_2ND_CLAMP4.Visu_Ret_Arr[5] := FALSE;
   S703_LM_DC_2ND_CLAMP4.Visu_Ret_Arr[6] := FALSE;
   S703_LM_DC_2ND_CLAMP4.Visu_Ret_Arr[7] := FALSE;
   S703_LM_DC_2ND_CLAMP4.Visu_Ret_Arr[8] := FALSE;
   S703_LM_DC_2ND_CLAMP4.Visu_Ret_Arr[9] := FALSE;
   S703_LM_DC_2ND_CLAMP4.Visu_Ret_Arr[10] := FALSE;
   S703_LM_DC_2ND_CLAMP4.Visu_Ret_Arr[11] := FALSE;
   S703_LM_DC_2ND_CLAMP4.Visu_Ret_Arr[12] := FALSE;
   S703_LM_DC_2ND_CLAMP4.Visu_Ret_Arr[13] := FALSE;
   S703_LM_DC_2ND_CLAMP4.Visu_Ret_Arr[14] := FALSE;
   S703_LM_DC_2ND_CLAMP4.Visu_Ret_Arr[15] := FALSE;
   S703_LM_DC_2ND_CLAMP4.BLK_Move_Ret := 0;
   S703_LM_DC_2ND_CLAMP4.Enable := FALSE;
   S703_LM_DC_2ND_CLAMP4.Adv_End := FALSE;
   S703_LM_DC_2ND_CLAMP4.Ret_End := FALSE;
   S703_LM_DC_2ND_CLAMP5.Enable_Aux := FALSE;
   S703_LM_DC_2ND_CLAMP5.Adv_Amount := 0;
   S703_LM_DC_2ND_CLAMP5.Ret_Amount := 0;
   S703_LM_DC_2ND_CLAMP5.LS_Adv1 := FALSE;
   S703_LM_DC_2ND_CLAMP5.LS_Ret1 := FALSE;
   S703_LM_DC_2ND_CLAMP5.LS_Adv2 := FALSE;
   S703_LM_DC_2ND_CLAMP5.LS_Ret2 := FALSE;
   S703_LM_DC_2ND_CLAMP5.LS_Adv3 := FALSE;
   S703_LM_DC_2ND_CLAMP5.LS_Ret3 := FALSE;
   S703_LM_DC_2ND_CLAMP5.LS_Adv4 := FALSE;
   S703_LM_DC_2ND_CLAMP5.LS_Ret4 := FALSE;
   S703_LM_DC_2ND_CLAMP5.SOL_Adv := FALSE;
   S703_LM_DC_2ND_CLAMP5.SOL_Ret := FALSE;
   S703_LM_DC_2ND_CLAMP5.M_Ready := FALSE;
   S703_LM_DC_2ND_CLAMP5.T_CHK1 := T#0MS;
   S703_LM_DC_2ND_CLAMP5.T_CHK2 := T#0MS;
   S703_LM_DC_2ND_CLAMP5.PB_Lamp_CHK := FALSE;
   S703_LM_DC_2ND_CLAMP5.PB_Error_Rst := FALSE;
   S703_LM_DC_2ND_CLAMP5.M_FLICK := FALSE;
   S703_LM_DC_2ND_CLAMP5.M_Adv_Err := FALSE;
   S703_LM_DC_2ND_CLAMP5.M_Ret_Err := FALSE;
   S703_LM_DC_2ND_CLAMP5.LP_Adv := FALSE;
   S703_LM_DC_2ND_CLAMP5.LP_Ret := FALSE;
   S703_LM_DC_2ND_CLAMP5.Visu_Adv := W#16#0;
   S703_LM_DC_2ND_CLAMP5.Visu_Ret := W#16#0;
   S703_LM_DC_2ND_CLAMP5.Error_T1.IN := FALSE;
   S703_LM_DC_2ND_CLAMP5.Error_T1.PT := T#0MS;
   S703_LM_DC_2ND_CLAMP5.Error_T1.Q := FALSE;
   S703_LM_DC_2ND_CLAMP5.Error_T1.ET := T#0MS;
   S703_LM_DC_2ND_CLAMP5.Error_T1.STATE := B#16#0;
   S703_LM_DC_2ND_CLAMP5.Error_T1.STIME := T#0MS;
   S703_LM_DC_2ND_CLAMP5.Error_T1.ATIME := T#0MS;
   S703_LM_DC_2ND_CLAMP5.Error_T2.IN := FALSE;
   S703_LM_DC_2ND_CLAMP5.Error_T2.PT := T#0MS;
   S703_LM_DC_2ND_CLAMP5.Error_T2.Q := FALSE;
   S703_LM_DC_2ND_CLAMP5.Error_T2.ET := T#0MS;
   S703_LM_DC_2ND_CLAMP5.Error_T2.STATE := B#16#0;
   S703_LM_DC_2ND_CLAMP5.Error_T2.STIME := T#0MS;
   S703_LM_DC_2ND_CLAMP5.Error_T2.ATIME := T#0MS;
   S703_LM_DC_2ND_CLAMP5.CHK_Aux1 := FALSE;
   S703_LM_DC_2ND_CLAMP5.CHK_Aux2 := FALSE;
   S703_LM_DC_2ND_CLAMP5.Error_T1_DN := FALSE;
   S703_LM_DC_2ND_CLAMP5.Error_T2_DN := FALSE;
   S703_LM_DC_2ND_CLAMP5.Adv_Memo := FALSE;
   S703_LM_DC_2ND_CLAMP5.Visu_Adv_Arr[0] := FALSE;
   S703_LM_DC_2ND_CLAMP5.Visu_Adv_Arr[1] := FALSE;
   S703_LM_DC_2ND_CLAMP5.Visu_Adv_Arr[2] := FALSE;
   S703_LM_DC_2ND_CLAMP5.Visu_Adv_Arr[3] := FALSE;
   S703_LM_DC_2ND_CLAMP5.Visu_Adv_Arr[4] := FALSE;
   S703_LM_DC_2ND_CLAMP5.Visu_Adv_Arr[5] := FALSE;
   S703_LM_DC_2ND_CLAMP5.Visu_Adv_Arr[6] := FALSE;
   S703_LM_DC_2ND_CLAMP5.Visu_Adv_Arr[7] := FALSE;
   S703_LM_DC_2ND_CLAMP5.Visu_Adv_Arr[8] := FALSE;
   S703_LM_DC_2ND_CLAMP5.Visu_Adv_Arr[9] := FALSE;
   S703_LM_DC_2ND_CLAMP5.Visu_Adv_Arr[10] := FALSE;
   S703_LM_DC_2ND_CLAMP5.Visu_Adv_Arr[11] := FALSE;
   S703_LM_DC_2ND_CLAMP5.Visu_Adv_Arr[12] := FALSE;
   S703_LM_DC_2ND_CLAMP5.Visu_Adv_Arr[13] := FALSE;
   S703_LM_DC_2ND_CLAMP5.Visu_Adv_Arr[14] := FALSE;
   S703_LM_DC_2ND_CLAMP5.Visu_Adv_Arr[15] := FALSE;
   S703_LM_DC_2ND_CLAMP5.Visu_Ret_Arr[0] := FALSE;
   S703_LM_DC_2ND_CLAMP5.Visu_Ret_Arr[1] := FALSE;
   S703_LM_DC_2ND_CLAMP5.Visu_Ret_Arr[2] := FALSE;
   S703_LM_DC_2ND_CLAMP5.Visu_Ret_Arr[3] := FALSE;
   S703_LM_DC_2ND_CLAMP5.Visu_Ret_Arr[4] := FALSE;
   S703_LM_DC_2ND_CLAMP5.Visu_Ret_Arr[5] := FALSE;
   S703_LM_DC_2ND_CLAMP5.Visu_Ret_Arr[6] := FALSE;
   S703_LM_DC_2ND_CLAMP5.Visu_Ret_Arr[7] := FALSE;
   S703_LM_DC_2ND_CLAMP5.Visu_Ret_Arr[8] := FALSE;
   S703_LM_DC_2ND_CLAMP5.Visu_Ret_Arr[9] := FALSE;
   S703_LM_DC_2ND_CLAMP5.Visu_Ret_Arr[10] := FALSE;
   S703_LM_DC_2ND_CLAMP5.Visu_Ret_Arr[11] := FALSE;
   S703_LM_DC_2ND_CLAMP5.Visu_Ret_Arr[12] := FALSE;
   S703_LM_DC_2ND_CLAMP5.Visu_Ret_Arr[13] := FALSE;
   S703_LM_DC_2ND_CLAMP5.Visu_Ret_Arr[14] := FALSE;
   S703_LM_DC_2ND_CLAMP5.Visu_Ret_Arr[15] := FALSE;
   S703_LM_DC_2ND_CLAMP5.BLK_Move_Ret := 0;
   S703_LM_DC_2ND_CLAMP5.Enable := FALSE;
   S703_LM_DC_2ND_CLAMP5.Adv_End := FALSE;
   S703_LM_DC_2ND_CLAMP5.Ret_End := FALSE;
   S703_LM_DC_STK_PIN.Enable_Aux := FALSE;
   S703_LM_DC_STK_PIN.Adv_Amount := 0;
   S703_LM_DC_STK_PIN.Ret_Amount := 0;
   S703_LM_DC_STK_PIN.LS_Adv1 := FALSE;
   S703_LM_DC_STK_PIN.LS_Ret1 := FALSE;
   S703_LM_DC_STK_PIN.LS_Adv2 := FALSE;
   S703_LM_DC_STK_PIN.LS_Ret2 := FALSE;
   S703_LM_DC_STK_PIN.LS_Adv3 := FALSE;
   S703_LM_DC_STK_PIN.LS_Ret3 := FALSE;
   S703_LM_DC_STK_PIN.LS_Adv4 := FALSE;
   S703_LM_DC_STK_PIN.LS_Ret4 := FALSE;
   S703_LM_DC_STK_PIN.SOL_Adv := FALSE;
   S703_LM_DC_STK_PIN.SOL_Ret := FALSE;
   S703_LM_DC_STK_PIN.M_Ready := FALSE;
   S703_LM_DC_STK_PIN.T_CHK1 := T#0MS;
   S703_LM_DC_STK_PIN.T_CHK2 := T#0MS;
   S703_LM_DC_STK_PIN.PB_Lamp_CHK := FALSE;
   S703_LM_DC_STK_PIN.PB_Error_Rst := FALSE;
   S703_LM_DC_STK_PIN.M_FLICK := FALSE;
   S703_LM_DC_STK_PIN.M_Adv_Err := FALSE;
   S703_LM_DC_STK_PIN.M_Ret_Err := FALSE;
   S703_LM_DC_STK_PIN.LP_Adv := FALSE;
   S703_LM_DC_STK_PIN.LP_Ret := FALSE;
   S703_LM_DC_STK_PIN.Visu_Adv := W#16#0;
   S703_LM_DC_STK_PIN.Visu_Ret := W#16#0;
   S703_LM_DC_STK_PIN.Error_T1.IN := FALSE;
   S703_LM_DC_STK_PIN.Error_T1.PT := T#0MS;
   S703_LM_DC_STK_PIN.Error_T1.Q := FALSE;
   S703_LM_DC_STK_PIN.Error_T1.ET := T#0MS;
   S703_LM_DC_STK_PIN.Error_T1.STATE := B#16#0;
   S703_LM_DC_STK_PIN.Error_T1.STIME := T#0MS;
   S703_LM_DC_STK_PIN.Error_T1.ATIME := T#0MS;
   S703_LM_DC_STK_PIN.Error_T2.IN := FALSE;
   S703_LM_DC_STK_PIN.Error_T2.PT := T#0MS;
   S703_LM_DC_STK_PIN.Error_T2.Q := FALSE;
   S703_LM_DC_STK_PIN.Error_T2.ET := T#0MS;
   S703_LM_DC_STK_PIN.Error_T2.STATE := B#16#0;
   S703_LM_DC_STK_PIN.Error_T2.STIME := T#0MS;
   S703_LM_DC_STK_PIN.Error_T2.ATIME := T#0MS;
   S703_LM_DC_STK_PIN.CHK_Aux1 := FALSE;
   S703_LM_DC_STK_PIN.CHK_Aux2 := FALSE;
   S703_LM_DC_STK_PIN.Error_T1_DN := FALSE;
   S703_LM_DC_STK_PIN.Error_T2_DN := FALSE;
   S703_LM_DC_STK_PIN.Adv_Memo := FALSE;
   S703_LM_DC_STK_PIN.Visu_Adv_Arr[0] := FALSE;
   S703_LM_DC_STK_PIN.Visu_Adv_Arr[1] := FALSE;
   S703_LM_DC_STK_PIN.Visu_Adv_Arr[2] := FALSE;
   S703_LM_DC_STK_PIN.Visu_Adv_Arr[3] := FALSE;
   S703_LM_DC_STK_PIN.Visu_Adv_Arr[4] := FALSE;
   S703_LM_DC_STK_PIN.Visu_Adv_Arr[5] := FALSE;
   S703_LM_DC_STK_PIN.Visu_Adv_Arr[6] := FALSE;
   S703_LM_DC_STK_PIN.Visu_Adv_Arr[7] := FALSE;
   S703_LM_DC_STK_PIN.Visu_Adv_Arr[8] := FALSE;
   S703_LM_DC_STK_PIN.Visu_Adv_Arr[9] := FALSE;
   S703_LM_DC_STK_PIN.Visu_Adv_Arr[10] := FALSE;
   S703_LM_DC_STK_PIN.Visu_Adv_Arr[11] := FALSE;
   S703_LM_DC_STK_PIN.Visu_Adv_Arr[12] := FALSE;
   S703_LM_DC_STK_PIN.Visu_Adv_Arr[13] := FALSE;
   S703_LM_DC_STK_PIN.Visu_Adv_Arr[14] := FALSE;
   S703_LM_DC_STK_PIN.Visu_Adv_Arr[15] := FALSE;
   S703_LM_DC_STK_PIN.Visu_Ret_Arr[0] := FALSE;
   S703_LM_DC_STK_PIN.Visu_Ret_Arr[1] := FALSE;
   S703_LM_DC_STK_PIN.Visu_Ret_Arr[2] := FALSE;
   S703_LM_DC_STK_PIN.Visu_Ret_Arr[3] := FALSE;
   S703_LM_DC_STK_PIN.Visu_Ret_Arr[4] := FALSE;
   S703_LM_DC_STK_PIN.Visu_Ret_Arr[5] := FALSE;
   S703_LM_DC_STK_PIN.Visu_Ret_Arr[6] := FALSE;
   S703_LM_DC_STK_PIN.Visu_Ret_Arr[7] := FALSE;
   S703_LM_DC_STK_PIN.Visu_Ret_Arr[8] := FALSE;
   S703_LM_DC_STK_PIN.Visu_Ret_Arr[9] := FALSE;
   S703_LM_DC_STK_PIN.Visu_Ret_Arr[10] := FALSE;
   S703_LM_DC_STK_PIN.Visu_Ret_Arr[11] := FALSE;
   S703_LM_DC_STK_PIN.Visu_Ret_Arr[12] := FALSE;
   S703_LM_DC_STK_PIN.Visu_Ret_Arr[13] := FALSE;
   S703_LM_DC_STK_PIN.Visu_Ret_Arr[14] := FALSE;
   S703_LM_DC_STK_PIN.Visu_Ret_Arr[15] := FALSE;
   S703_LM_DC_STK_PIN.BLK_Move_Ret := 0;
   S703_LM_DC_STK_PIN.Enable := FALSE;
   S703_LM_DC_STK_PIN.Adv_End := FALSE;
   S703_LM_DC_STK_PIN.Ret_End := FALSE;
   S703_LM_DC_OTR_CLAMP.Enable_Aux := FALSE;
   S703_LM_DC_OTR_CLAMP.Adv_Amount := 0;
   S703_LM_DC_OTR_CLAMP.Ret_Amount := 0;
   S703_LM_DC_OTR_CLAMP.LS_Adv1 := FALSE;
   S703_LM_DC_OTR_CLAMP.LS_Ret1 := FALSE;
   S703_LM_DC_OTR_CLAMP.LS_Adv2 := FALSE;
   S703_LM_DC_OTR_CLAMP.LS_Ret2 := FALSE;
   S703_LM_DC_OTR_CLAMP.LS_Adv3 := FALSE;
   S703_LM_DC_OTR_CLAMP.LS_Ret3 := FALSE;
   S703_LM_DC_OTR_CLAMP.LS_Adv4 := FALSE;
   S703_LM_DC_OTR_CLAMP.LS_Ret4 := FALSE;
   S703_LM_DC_OTR_CLAMP.SOL_Adv := FALSE;
   S703_LM_DC_OTR_CLAMP.SOL_Ret := FALSE;
   S703_LM_DC_OTR_CLAMP.M_Ready := FALSE;
   S703_LM_DC_OTR_CLAMP.T_CHK1 := T#0MS;
   S703_LM_DC_OTR_CLAMP.T_CHK2 := T#0MS;
   S703_LM_DC_OTR_CLAMP.PB_Lamp_CHK := FALSE;
   S703_LM_DC_OTR_CLAMP.PB_Error_Rst := FALSE;
   S703_LM_DC_OTR_CLAMP.M_FLICK := FALSE;
   S703_LM_DC_OTR_CLAMP.M_Adv_Err := FALSE;
   S703_LM_DC_OTR_CLAMP.M_Ret_Err := FALSE;
   S703_LM_DC_OTR_CLAMP.LP_Adv := FALSE;
   S703_LM_DC_OTR_CLAMP.LP_Ret := FALSE;
   S703_LM_DC_OTR_CLAMP.Visu_Adv := W#16#0;
   S703_LM_DC_OTR_CLAMP.Visu_Ret := W#16#0;
   S703_LM_DC_OTR_CLAMP.Error_T1.IN := FALSE;
   S703_LM_DC_OTR_CLAMP.Error_T1.PT := T#0MS;
   S703_LM_DC_OTR_CLAMP.Error_T1.Q := FALSE;
   S703_LM_DC_OTR_CLAMP.Error_T1.ET := T#0MS;
   S703_LM_DC_OTR_CLAMP.Error_T1.STATE := B#16#0;
   S703_LM_DC_OTR_CLAMP.Error_T1.STIME := T#0MS;
   S703_LM_DC_OTR_CLAMP.Error_T1.ATIME := T#0MS;
   S703_LM_DC_OTR_CLAMP.Error_T2.IN := FALSE;
   S703_LM_DC_OTR_CLAMP.Error_T2.PT := T#0MS;
   S703_LM_DC_OTR_CLAMP.Error_T2.Q := FALSE;
   S703_LM_DC_OTR_CLAMP.Error_T2.ET := T#0MS;
   S703_LM_DC_OTR_CLAMP.Error_T2.STATE := B#16#0;
   S703_LM_DC_OTR_CLAMP.Error_T2.STIME := T#0MS;
   S703_LM_DC_OTR_CLAMP.Error_T2.ATIME := T#0MS;
   S703_LM_DC_OTR_CLAMP.CHK_Aux1 := FALSE;
   S703_LM_DC_OTR_CLAMP.CHK_Aux2 := FALSE;
   S703_LM_DC_OTR_CLAMP.Error_T1_DN := FALSE;
   S703_LM_DC_OTR_CLAMP.Error_T2_DN := FALSE;
   S703_LM_DC_OTR_CLAMP.Adv_Memo := FALSE;
   S703_LM_DC_OTR_CLAMP.Visu_Adv_Arr[0] := FALSE;
   S703_LM_DC_OTR_CLAMP.Visu_Adv_Arr[1] := FALSE;
   S703_LM_DC_OTR_CLAMP.Visu_Adv_Arr[2] := FALSE;
   S703_LM_DC_OTR_CLAMP.Visu_Adv_Arr[3] := FALSE;
   S703_LM_DC_OTR_CLAMP.Visu_Adv_Arr[4] := FALSE;
   S703_LM_DC_OTR_CLAMP.Visu_Adv_Arr[5] := FALSE;
   S703_LM_DC_OTR_CLAMP.Visu_Adv_Arr[6] := FALSE;
   S703_LM_DC_OTR_CLAMP.Visu_Adv_Arr[7] := FALSE;
   S703_LM_DC_OTR_CLAMP.Visu_Adv_Arr[8] := FALSE;
   S703_LM_DC_OTR_CLAMP.Visu_Adv_Arr[9] := FALSE;
   S703_LM_DC_OTR_CLAMP.Visu_Adv_Arr[10] := FALSE;
   S703_LM_DC_OTR_CLAMP.Visu_Adv_Arr[11] := FALSE;
   S703_LM_DC_OTR_CLAMP.Visu_Adv_Arr[12] := FALSE;
   S703_LM_DC_OTR_CLAMP.Visu_Adv_Arr[13] := FALSE;
   S703_LM_DC_OTR_CLAMP.Visu_Adv_Arr[14] := FALSE;
   S703_LM_DC_OTR_CLAMP.Visu_Adv_Arr[15] := FALSE;
   S703_LM_DC_OTR_CLAMP.Visu_Ret_Arr[0] := FALSE;
   S703_LM_DC_OTR_CLAMP.Visu_Ret_Arr[1] := FALSE;
   S703_LM_DC_OTR_CLAMP.Visu_Ret_Arr[2] := FALSE;
   S703_LM_DC_OTR_CLAMP.Visu_Ret_Arr[3] := FALSE;
   S703_LM_DC_OTR_CLAMP.Visu_Ret_Arr[4] := FALSE;
   S703_LM_DC_OTR_CLAMP.Visu_Ret_Arr[5] := FALSE;
   S703_LM_DC_OTR_CLAMP.Visu_Ret_Arr[6] := FALSE;
   S703_LM_DC_OTR_CLAMP.Visu_Ret_Arr[7] := FALSE;
   S703_LM_DC_OTR_CLAMP.Visu_Ret_Arr[8] := FALSE;
   S703_LM_DC_OTR_CLAMP.Visu_Ret_Arr[9] := FALSE;
   S703_LM_DC_OTR_CLAMP.Visu_Ret_Arr[10] := FALSE;
   S703_LM_DC_OTR_CLAMP.Visu_Ret_Arr[11] := FALSE;
   S703_LM_DC_OTR_CLAMP.Visu_Ret_Arr[12] := FALSE;
   S703_LM_DC_OTR_CLAMP.Visu_Ret_Arr[13] := FALSE;
   S703_LM_DC_OTR_CLAMP.Visu_Ret_Arr[14] := FALSE;
   S703_LM_DC_OTR_CLAMP.Visu_Ret_Arr[15] := FALSE;
   S703_LM_DC_OTR_CLAMP.BLK_Move_Ret := 0;
   S703_LM_DC_OTR_CLAMP.Enable := FALSE;
   S703_LM_DC_OTR_CLAMP.Adv_End := FALSE;
   S703_LM_DC_OTR_CLAMP.Ret_End := FALSE;
   S703_LM_DC_ASSY_CLAMP.Enable_Aux := FALSE;
   S703_LM_DC_ASSY_CLAMP.Adv_Amount := 0;
   S703_LM_DC_ASSY_CLAMP.Ret_Amount := 0;
   S703_LM_DC_ASSY_CLAMP.LS_Adv1 := FALSE;
   S703_LM_DC_ASSY_CLAMP.LS_Ret1 := FALSE;
   S703_LM_DC_ASSY_CLAMP.LS_Adv2 := FALSE;
   S703_LM_DC_ASSY_CLAMP.LS_Ret2 := FALSE;
   S703_LM_DC_ASSY_CLAMP.LS_Adv3 := FALSE;
   S703_LM_DC_ASSY_CLAMP.LS_Ret3 := FALSE;
   S703_LM_DC_ASSY_CLAMP.LS_Adv4 := FALSE;
   S703_LM_DC_ASSY_CLAMP.LS_Ret4 := FALSE;
   S703_LM_DC_ASSY_CLAMP.SOL_Adv := FALSE;
   S703_LM_DC_ASSY_CLAMP.SOL_Ret := FALSE;
   S703_LM_DC_ASSY_CLAMP.M_Ready := FALSE;
   S703_LM_DC_ASSY_CLAMP.T_CHK1 := T#0MS;
   S703_LM_DC_ASSY_CLAMP.T_CHK2 := T#0MS;
   S703_LM_DC_ASSY_CLAMP.PB_Lamp_CHK := FALSE;
   S703_LM_DC_ASSY_CLAMP.PB_Error_Rst := FALSE;
   S703_LM_DC_ASSY_CLAMP.M_FLICK := FALSE;
   S703_LM_DC_ASSY_CLAMP.M_Adv_Err := FALSE;
   S703_LM_DC_ASSY_CLAMP.M_Ret_Err := FALSE;
   S703_LM_DC_ASSY_CLAMP.LP_Adv := FALSE;
   S703_LM_DC_ASSY_CLAMP.LP_Ret := FALSE;
   S703_LM_DC_ASSY_CLAMP.Visu_Adv := W#16#0;
   S703_LM_DC_ASSY_CLAMP.Visu_Ret := W#16#0;
   S703_LM_DC_ASSY_CLAMP.Error_T1.IN := FALSE;
   S703_LM_DC_ASSY_CLAMP.Error_T1.PT := T#0MS;
   S703_LM_DC_ASSY_CLAMP.Error_T1.Q := FALSE;
   S703_LM_DC_ASSY_CLAMP.Error_T1.ET := T#0MS;
   S703_LM_DC_ASSY_CLAMP.Error_T1.STATE := B#16#0;
   S703_LM_DC_ASSY_CLAMP.Error_T1.STIME := T#0MS;
   S703_LM_DC_ASSY_CLAMP.Error_T1.ATIME := T#0MS;
   S703_LM_DC_ASSY_CLAMP.Error_T2.IN := FALSE;
   S703_LM_DC_ASSY_CLAMP.Error_T2.PT := T#0MS;
   S703_LM_DC_ASSY_CLAMP.Error_T2.Q := FALSE;
   S703_LM_DC_ASSY_CLAMP.Error_T2.ET := T#0MS;
   S703_LM_DC_ASSY_CLAMP.Error_T2.STATE := B#16#0;
   S703_LM_DC_ASSY_CLAMP.Error_T2.STIME := T#0MS;
   S703_LM_DC_ASSY_CLAMP.Error_T2.ATIME := T#0MS;
   S703_LM_DC_ASSY_CLAMP.CHK_Aux1 := FALSE;
   S703_LM_DC_ASSY_CLAMP.CHK_Aux2 := FALSE;
   S703_LM_DC_ASSY_CLAMP.Error_T1_DN := FALSE;
   S703_LM_DC_ASSY_CLAMP.Error_T2_DN := FALSE;
   S703_LM_DC_ASSY_CLAMP.Adv_Memo := FALSE;
   S703_LM_DC_ASSY_CLAMP.Visu_Adv_Arr[0] := FALSE;
   S703_LM_DC_ASSY_CLAMP.Visu_Adv_Arr[1] := FALSE;
   S703_LM_DC_ASSY_CLAMP.Visu_Adv_Arr[2] := FALSE;
   S703_LM_DC_ASSY_CLAMP.Visu_Adv_Arr[3] := FALSE;
   S703_LM_DC_ASSY_CLAMP.Visu_Adv_Arr[4] := FALSE;
   S703_LM_DC_ASSY_CLAMP.Visu_Adv_Arr[5] := FALSE;
   S703_LM_DC_ASSY_CLAMP.Visu_Adv_Arr[6] := FALSE;
   S703_LM_DC_ASSY_CLAMP.Visu_Adv_Arr[7] := FALSE;
   S703_LM_DC_ASSY_CLAMP.Visu_Adv_Arr[8] := FALSE;
   S703_LM_DC_ASSY_CLAMP.Visu_Adv_Arr[9] := FALSE;
   S703_LM_DC_ASSY_CLAMP.Visu_Adv_Arr[10] := FALSE;
   S703_LM_DC_ASSY_CLAMP.Visu_Adv_Arr[11] := FALSE;
   S703_LM_DC_ASSY_CLAMP.Visu_Adv_Arr[12] := FALSE;
   S703_LM_DC_ASSY_CLAMP.Visu_Adv_Arr[13] := FALSE;
   S703_LM_DC_ASSY_CLAMP.Visu_Adv_Arr[14] := FALSE;
   S703_LM_DC_ASSY_CLAMP.Visu_Adv_Arr[15] := FALSE;
   S703_LM_DC_ASSY_CLAMP.Visu_Ret_Arr[0] := FALSE;
   S703_LM_DC_ASSY_CLAMP.Visu_Ret_Arr[1] := FALSE;
   S703_LM_DC_ASSY_CLAMP.Visu_Ret_Arr[2] := FALSE;
   S703_LM_DC_ASSY_CLAMP.Visu_Ret_Arr[3] := FALSE;
   S703_LM_DC_ASSY_CLAMP.Visu_Ret_Arr[4] := FALSE;
   S703_LM_DC_ASSY_CLAMP.Visu_Ret_Arr[5] := FALSE;
   S703_LM_DC_ASSY_CLAMP.Visu_Ret_Arr[6] := FALSE;
   S703_LM_DC_ASSY_CLAMP.Visu_Ret_Arr[7] := FALSE;
   S703_LM_DC_ASSY_CLAMP.Visu_Ret_Arr[8] := FALSE;
   S703_LM_DC_ASSY_CLAMP.Visu_Ret_Arr[9] := FALSE;
   S703_LM_DC_ASSY_CLAMP.Visu_Ret_Arr[10] := FALSE;
   S703_LM_DC_ASSY_CLAMP.Visu_Ret_Arr[11] := FALSE;
   S703_LM_DC_ASSY_CLAMP.Visu_Ret_Arr[12] := FALSE;
   S703_LM_DC_ASSY_CLAMP.Visu_Ret_Arr[13] := FALSE;
   S703_LM_DC_ASSY_CLAMP.Visu_Ret_Arr[14] := FALSE;
   S703_LM_DC_ASSY_CLAMP.Visu_Ret_Arr[15] := FALSE;
   S703_LM_DC_ASSY_CLAMP.BLK_Move_Ret := 0;
   S703_LM_DC_ASSY_CLAMP.Enable := FALSE;
   S703_LM_DC_ASSY_CLAMP.Adv_End := FALSE;
   S703_LM_DC_ASSY_CLAMP.Ret_End := FALSE;
   S703_LM_DC_FF_PIN.Enable_Aux := FALSE;
   S703_LM_DC_FF_PIN.Adv_Amount := 0;
   S703_LM_DC_FF_PIN.Ret_Amount := 0;
   S703_LM_DC_FF_PIN.LS_Adv1 := FALSE;
   S703_LM_DC_FF_PIN.LS_Ret1 := FALSE;
   S703_LM_DC_FF_PIN.LS_Adv2 := FALSE;
   S703_LM_DC_FF_PIN.LS_Ret2 := FALSE;
   S703_LM_DC_FF_PIN.LS_Adv3 := FALSE;
   S703_LM_DC_FF_PIN.LS_Ret3 := FALSE;
   S703_LM_DC_FF_PIN.LS_Adv4 := FALSE;
   S703_LM_DC_FF_PIN.LS_Ret4 := FALSE;
   S703_LM_DC_FF_PIN.SOL_Adv := FALSE;
   S703_LM_DC_FF_PIN.SOL_Ret := FALSE;
   S703_LM_DC_FF_PIN.M_Ready := FALSE;
   S703_LM_DC_FF_PIN.T_CHK1 := T#0MS;
   S703_LM_DC_FF_PIN.T_CHK2 := T#0MS;
   S703_LM_DC_FF_PIN.PB_Lamp_CHK := FALSE;
   S703_LM_DC_FF_PIN.PB_Error_Rst := FALSE;
   S703_LM_DC_FF_PIN.M_FLICK := FALSE;
   S703_LM_DC_FF_PIN.M_Adv_Err := FALSE;
   S703_LM_DC_FF_PIN.M_Ret_Err := FALSE;
   S703_LM_DC_FF_PIN.LP_Adv := FALSE;
   S703_LM_DC_FF_PIN.LP_Ret := FALSE;
   S703_LM_DC_FF_PIN.Visu_Adv := W#16#0;
   S703_LM_DC_FF_PIN.Visu_Ret := W#16#0;
   S703_LM_DC_FF_PIN.Error_T1.IN := FALSE;
   S703_LM_DC_FF_PIN.Error_T1.PT := T#0MS;
   S703_LM_DC_FF_PIN.Error_T1.Q := FALSE;
   S703_LM_DC_FF_PIN.Error_T1.ET := T#0MS;
   S703_LM_DC_FF_PIN.Error_T1.STATE := B#16#0;
   S703_LM_DC_FF_PIN.Error_T1.STIME := T#0MS;
   S703_LM_DC_FF_PIN.Error_T1.ATIME := T#0MS;
   S703_LM_DC_FF_PIN.Error_T2.IN := FALSE;
   S703_LM_DC_FF_PIN.Error_T2.PT := T#0MS;
   S703_LM_DC_FF_PIN.Error_T2.Q := FALSE;
   S703_LM_DC_FF_PIN.Error_T2.ET := T#0MS;
   S703_LM_DC_FF_PIN.Error_T2.STATE := B#16#0;
   S703_LM_DC_FF_PIN.Error_T2.STIME := T#0MS;
   S703_LM_DC_FF_PIN.Error_T2.ATIME := T#0MS;
   S703_LM_DC_FF_PIN.CHK_Aux1 := FALSE;
   S703_LM_DC_FF_PIN.CHK_Aux2 := FALSE;
   S703_LM_DC_FF_PIN.Error_T1_DN := FALSE;
   S703_LM_DC_FF_PIN.Error_T2_DN := FALSE;
   S703_LM_DC_FF_PIN.Adv_Memo := FALSE;
   S703_LM_DC_FF_PIN.Visu_Adv_Arr[0] := FALSE;
   S703_LM_DC_FF_PIN.Visu_Adv_Arr[1] := FALSE;
   S703_LM_DC_FF_PIN.Visu_Adv_Arr[2] := FALSE;
   S703_LM_DC_FF_PIN.Visu_Adv_Arr[3] := FALSE;
   S703_LM_DC_FF_PIN.Visu_Adv_Arr[4] := FALSE;
   S703_LM_DC_FF_PIN.Visu_Adv_Arr[5] := FALSE;
   S703_LM_DC_FF_PIN.Visu_Adv_Arr[6] := FALSE;
   S703_LM_DC_FF_PIN.Visu_Adv_Arr[7] := FALSE;
   S703_LM_DC_FF_PIN.Visu_Adv_Arr[8] := FALSE;
   S703_LM_DC_FF_PIN.Visu_Adv_Arr[9] := FALSE;
   S703_LM_DC_FF_PIN.Visu_Adv_Arr[10] := FALSE;
   S703_LM_DC_FF_PIN.Visu_Adv_Arr[11] := FALSE;
   S703_LM_DC_FF_PIN.Visu_Adv_Arr[12] := FALSE;
   S703_LM_DC_FF_PIN.Visu_Adv_Arr[13] := FALSE;
   S703_LM_DC_FF_PIN.Visu_Adv_Arr[14] := FALSE;
   S703_LM_DC_FF_PIN.Visu_Adv_Arr[15] := FALSE;
   S703_LM_DC_FF_PIN.Visu_Ret_Arr[0] := FALSE;
   S703_LM_DC_FF_PIN.Visu_Ret_Arr[1] := FALSE;
   S703_LM_DC_FF_PIN.Visu_Ret_Arr[2] := FALSE;
   S703_LM_DC_FF_PIN.Visu_Ret_Arr[3] := FALSE;
   S703_LM_DC_FF_PIN.Visu_Ret_Arr[4] := FALSE;
   S703_LM_DC_FF_PIN.Visu_Ret_Arr[5] := FALSE;
   S703_LM_DC_FF_PIN.Visu_Ret_Arr[6] := FALSE;
   S703_LM_DC_FF_PIN.Visu_Ret_Arr[7] := FALSE;
   S703_LM_DC_FF_PIN.Visu_Ret_Arr[8] := FALSE;
   S703_LM_DC_FF_PIN.Visu_Ret_Arr[9] := FALSE;
   S703_LM_DC_FF_PIN.Visu_Ret_Arr[10] := FALSE;
   S703_LM_DC_FF_PIN.Visu_Ret_Arr[11] := FALSE;
   S703_LM_DC_FF_PIN.Visu_Ret_Arr[12] := FALSE;
   S703_LM_DC_FF_PIN.Visu_Ret_Arr[13] := FALSE;
   S703_LM_DC_FF_PIN.Visu_Ret_Arr[14] := FALSE;
   S703_LM_DC_FF_PIN.Visu_Ret_Arr[15] := FALSE;
   S703_LM_DC_FF_PIN.BLK_Move_Ret := 0;
   S703_LM_DC_FF_PIN.Enable := FALSE;
   S703_LM_DC_FF_PIN.Adv_End := FALSE;
   S703_LM_DC_FF_PIN.Ret_End := FALSE;
   S703_LM_DC_FF_CLAMP.Enable_Aux := FALSE;
   S703_LM_DC_FF_CLAMP.Adv_Amount := 0;
   S703_LM_DC_FF_CLAMP.Ret_Amount := 0;
   S703_LM_DC_FF_CLAMP.LS_Adv1 := FALSE;
   S703_LM_DC_FF_CLAMP.LS_Ret1 := FALSE;
   S703_LM_DC_FF_CLAMP.LS_Adv2 := FALSE;
   S703_LM_DC_FF_CLAMP.LS_Ret2 := FALSE;
   S703_LM_DC_FF_CLAMP.LS_Adv3 := FALSE;
   S703_LM_DC_FF_CLAMP.LS_Ret3 := FALSE;
   S703_LM_DC_FF_CLAMP.LS_Adv4 := FALSE;
   S703_LM_DC_FF_CLAMP.LS_Ret4 := FALSE;
   S703_LM_DC_FF_CLAMP.SOL_Adv := FALSE;
   S703_LM_DC_FF_CLAMP.SOL_Ret := FALSE;
   S703_LM_DC_FF_CLAMP.M_Ready := FALSE;
   S703_LM_DC_FF_CLAMP.T_CHK1 := T#0MS;
   S703_LM_DC_FF_CLAMP.T_CHK2 := T#0MS;
   S703_LM_DC_FF_CLAMP.PB_Lamp_CHK := FALSE;
   S703_LM_DC_FF_CLAMP.PB_Error_Rst := FALSE;
   S703_LM_DC_FF_CLAMP.M_FLICK := FALSE;
   S703_LM_DC_FF_CLAMP.M_Adv_Err := FALSE;
   S703_LM_DC_FF_CLAMP.M_Ret_Err := FALSE;
   S703_LM_DC_FF_CLAMP.LP_Adv := FALSE;
   S703_LM_DC_FF_CLAMP.LP_Ret := FALSE;
   S703_LM_DC_FF_CLAMP.Visu_Adv := W#16#0;
   S703_LM_DC_FF_CLAMP.Visu_Ret := W#16#0;
   S703_LM_DC_FF_CLAMP.Error_T1.IN := FALSE;
   S703_LM_DC_FF_CLAMP.Error_T1.PT := T#0MS;
   S703_LM_DC_FF_CLAMP.Error_T1.Q := FALSE;
   S703_LM_DC_FF_CLAMP.Error_T1.ET := T#0MS;
   S703_LM_DC_FF_CLAMP.Error_T1.STATE := B#16#0;
   S703_LM_DC_FF_CLAMP.Error_T1.STIME := T#0MS;
   S703_LM_DC_FF_CLAMP.Error_T1.ATIME := T#0MS;
   S703_LM_DC_FF_CLAMP.Error_T2.IN := FALSE;
   S703_LM_DC_FF_CLAMP.Error_T2.PT := T#0MS;
   S703_LM_DC_FF_CLAMP.Error_T2.Q := FALSE;
   S703_LM_DC_FF_CLAMP.Error_T2.ET := T#0MS;
   S703_LM_DC_FF_CLAMP.Error_T2.STATE := B#16#0;
   S703_LM_DC_FF_CLAMP.Error_T2.STIME := T#0MS;
   S703_LM_DC_FF_CLAMP.Error_T2.ATIME := T#0MS;
   S703_LM_DC_FF_CLAMP.CHK_Aux1 := FALSE;
   S703_LM_DC_FF_CLAMP.CHK_Aux2 := FALSE;
   S703_LM_DC_FF_CLAMP.Error_T1_DN := FALSE;
   S703_LM_DC_FF_CLAMP.Error_T2_DN := FALSE;
   S703_LM_DC_FF_CLAMP.Adv_Memo := FALSE;
   S703_LM_DC_FF_CLAMP.Visu_Adv_Arr[0] := FALSE;
   S703_LM_DC_FF_CLAMP.Visu_Adv_Arr[1] := FALSE;
   S703_LM_DC_FF_CLAMP.Visu_Adv_Arr[2] := FALSE;
   S703_LM_DC_FF_CLAMP.Visu_Adv_Arr[3] := FALSE;
   S703_LM_DC_FF_CLAMP.Visu_Adv_Arr[4] := FALSE;
   S703_LM_DC_FF_CLAMP.Visu_Adv_Arr[5] := FALSE;
   S703_LM_DC_FF_CLAMP.Visu_Adv_Arr[6] := FALSE;
   S703_LM_DC_FF_CLAMP.Visu_Adv_Arr[7] := FALSE;
   S703_LM_DC_FF_CLAMP.Visu_Adv_Arr[8] := FALSE;
   S703_LM_DC_FF_CLAMP.Visu_Adv_Arr[9] := FALSE;
   S703_LM_DC_FF_CLAMP.Visu_Adv_Arr[10] := FALSE;
   S703_LM_DC_FF_CLAMP.Visu_Adv_Arr[11] := FALSE;
   S703_LM_DC_FF_CLAMP.Visu_Adv_Arr[12] := FALSE;
   S703_LM_DC_FF_CLAMP.Visu_Adv_Arr[13] := FALSE;
   S703_LM_DC_FF_CLAMP.Visu_Adv_Arr[14] := FALSE;
   S703_LM_DC_FF_CLAMP.Visu_Adv_Arr[15] := FALSE;
   S703_LM_DC_FF_CLAMP.Visu_Ret_Arr[0] := FALSE;
   S703_LM_DC_FF_CLAMP.Visu_Ret_Arr[1] := FALSE;
   S703_LM_DC_FF_CLAMP.Visu_Ret_Arr[2] := FALSE;
   S703_LM_DC_FF_CLAMP.Visu_Ret_Arr[3] := FALSE;
   S703_LM_DC_FF_CLAMP.Visu_Ret_Arr[4] := FALSE;
   S703_LM_DC_FF_CLAMP.Visu_Ret_Arr[5] := FALSE;
   S703_LM_DC_FF_CLAMP.Visu_Ret_Arr[6] := FALSE;
   S703_LM_DC_FF_CLAMP.Visu_Ret_Arr[7] := FALSE;
   S703_LM_DC_FF_CLAMP.Visu_Ret_Arr[8] := FALSE;
   S703_LM_DC_FF_CLAMP.Visu_Ret_Arr[9] := FALSE;
   S703_LM_DC_FF_CLAMP.Visu_Ret_Arr[10] := FALSE;
   S703_LM_DC_FF_CLAMP.Visu_Ret_Arr[11] := FALSE;
   S703_LM_DC_FF_CLAMP.Visu_Ret_Arr[12] := FALSE;
   S703_LM_DC_FF_CLAMP.Visu_Ret_Arr[13] := FALSE;
   S703_LM_DC_FF_CLAMP.Visu_Ret_Arr[14] := FALSE;
   S703_LM_DC_FF_CLAMP.Visu_Ret_Arr[15] := FALSE;
   S703_LM_DC_FF_CLAMP.BLK_Move_Ret := 0;
   S703_LM_DC_FF_CLAMP.Enable := FALSE;
   S703_LM_DC_FF_CLAMP.Adv_End := FALSE;
   S703_LM_DC_FF_CLAMP.Ret_End := FALSE;
   S703_LM_DC_2ND_CLAMP6.Enable_Aux := FALSE;
   S703_LM_DC_2ND_CLAMP6.Adv_Amount := 0;
   S703_LM_DC_2ND_CLAMP6.Ret_Amount := 0;
   S703_LM_DC_2ND_CLAMP6.LS_Adv1 := FALSE;
   S703_LM_DC_2ND_CLAMP6.LS_Ret1 := FALSE;
   S703_LM_DC_2ND_CLAMP6.LS_Adv2 := FALSE;
   S703_LM_DC_2ND_CLAMP6.LS_Ret2 := FALSE;
   S703_LM_DC_2ND_CLAMP6.LS_Adv3 := FALSE;
   S703_LM_DC_2ND_CLAMP6.LS_Ret3 := FALSE;
   S703_LM_DC_2ND_CLAMP6.LS_Adv4 := FALSE;
   S703_LM_DC_2ND_CLAMP6.LS_Ret4 := FALSE;
   S703_LM_DC_2ND_CLAMP6.SOL_Adv := FALSE;
   S703_LM_DC_2ND_CLAMP6.SOL_Ret := FALSE;
   S703_LM_DC_2ND_CLAMP6.M_Ready := FALSE;
   S703_LM_DC_2ND_CLAMP6.T_CHK1 := T#0MS;
   S703_LM_DC_2ND_CLAMP6.T_CHK2 := T#0MS;
   S703_LM_DC_2ND_CLAMP6.PB_Lamp_CHK := FALSE;
   S703_LM_DC_2ND_CLAMP6.PB_Error_Rst := FALSE;
   S703_LM_DC_2ND_CLAMP6.M_FLICK := FALSE;
   S703_LM_DC_2ND_CLAMP6.M_Adv_Err := FALSE;
   S703_LM_DC_2ND_CLAMP6.M_Ret_Err := FALSE;
   S703_LM_DC_2ND_CLAMP6.LP_Adv := FALSE;
   S703_LM_DC_2ND_CLAMP6.LP_Ret := FALSE;
   S703_LM_DC_2ND_CLAMP6.Visu_Adv := W#16#0;
   S703_LM_DC_2ND_CLAMP6.Visu_Ret := W#16#0;
   S703_LM_DC_2ND_CLAMP6.Error_T1.IN := FALSE;
   S703_LM_DC_2ND_CLAMP6.Error_T1.PT := T#0MS;
   S703_LM_DC_2ND_CLAMP6.Error_T1.Q := FALSE;
   S703_LM_DC_2ND_CLAMP6.Error_T1.ET := T#0MS;
   S703_LM_DC_2ND_CLAMP6.Error_T1.STATE := B#16#0;
   S703_LM_DC_2ND_CLAMP6.Error_T1.STIME := T#0MS;
   S703_LM_DC_2ND_CLAMP6.Error_T1.ATIME := T#0MS;
   S703_LM_DC_2ND_CLAMP6.Error_T2.IN := FALSE;
   S703_LM_DC_2ND_CLAMP6.Error_T2.PT := T#0MS;
   S703_LM_DC_2ND_CLAMP6.Error_T2.Q := FALSE;
